// TIA Portal V15.1 export
// export: Created 2024-05-17T05:38:54.9561831Z, ExportSetting WithDefaults, DisplayName Totally Integrated Automation Portal, DisplayVersion V15.1 Update 5, DisplayName TIA Portal Openness, DisplayVersion V15.1 Update 5, DisplayName SINAMICS Startdrive Advanced, DisplayVersion V15.1, DisplayName G130, G150, S120, S150, SINAMICS MV, S210, DisplayVersion V15.1, DisplayName G110M, G120, G120C, G120D, G120P, DisplayVersion V15.1, DisplayName STEP 7 Professional, DisplayVersion V15.1 Update 5, DisplayName STEP 7 Safety, DisplayVersion V15.1, DisplayName WinCC Professional, DisplayVersion V15.1 Update 5, DisplayName SIMATIC Visualization Architect, DisplayVersion V15.1
FUNCTION "209220ZM01" : Void   // FC350, FBD
TITLE = 209220ZM01 ModeZone
{ S7_Optimized_Access := 'FALSE' }
AUTHOR : VCG
NAME : Mot001
VERSION : 0.1
// stored: AutoNumber false, IsIECCheckEnabled false, SetENOAutomatically False, UDAEnableTagReadback false
   VAR_OUTPUT
      O_AlarmA : Bool;   // Alarm A
      O_AlarmB : Bool;   // Alarm B
      O_AlarmC : Bool;   // Alarm C
      O_AlarmD : Bool;   // Alarm D
      O_AlarmABCondition : Bool;   // Alarms resetable
      H_IAnim : Word;   // Animation bits to Icon in WinCC
   END_VAR
   VAR_TEMP
      TempReal : Real;
      TempInt : Int;
   END_VAR
   VAR_TEMP   // added for the SCL form of the ladder/FBD networks
      _w1 : Bool;
      _w2 : Bool;
   END_VAR
BEGIN

REGION Network 1: **** 1 - Inputs **** HMI Commands
   // HMI Commands from the WinCC
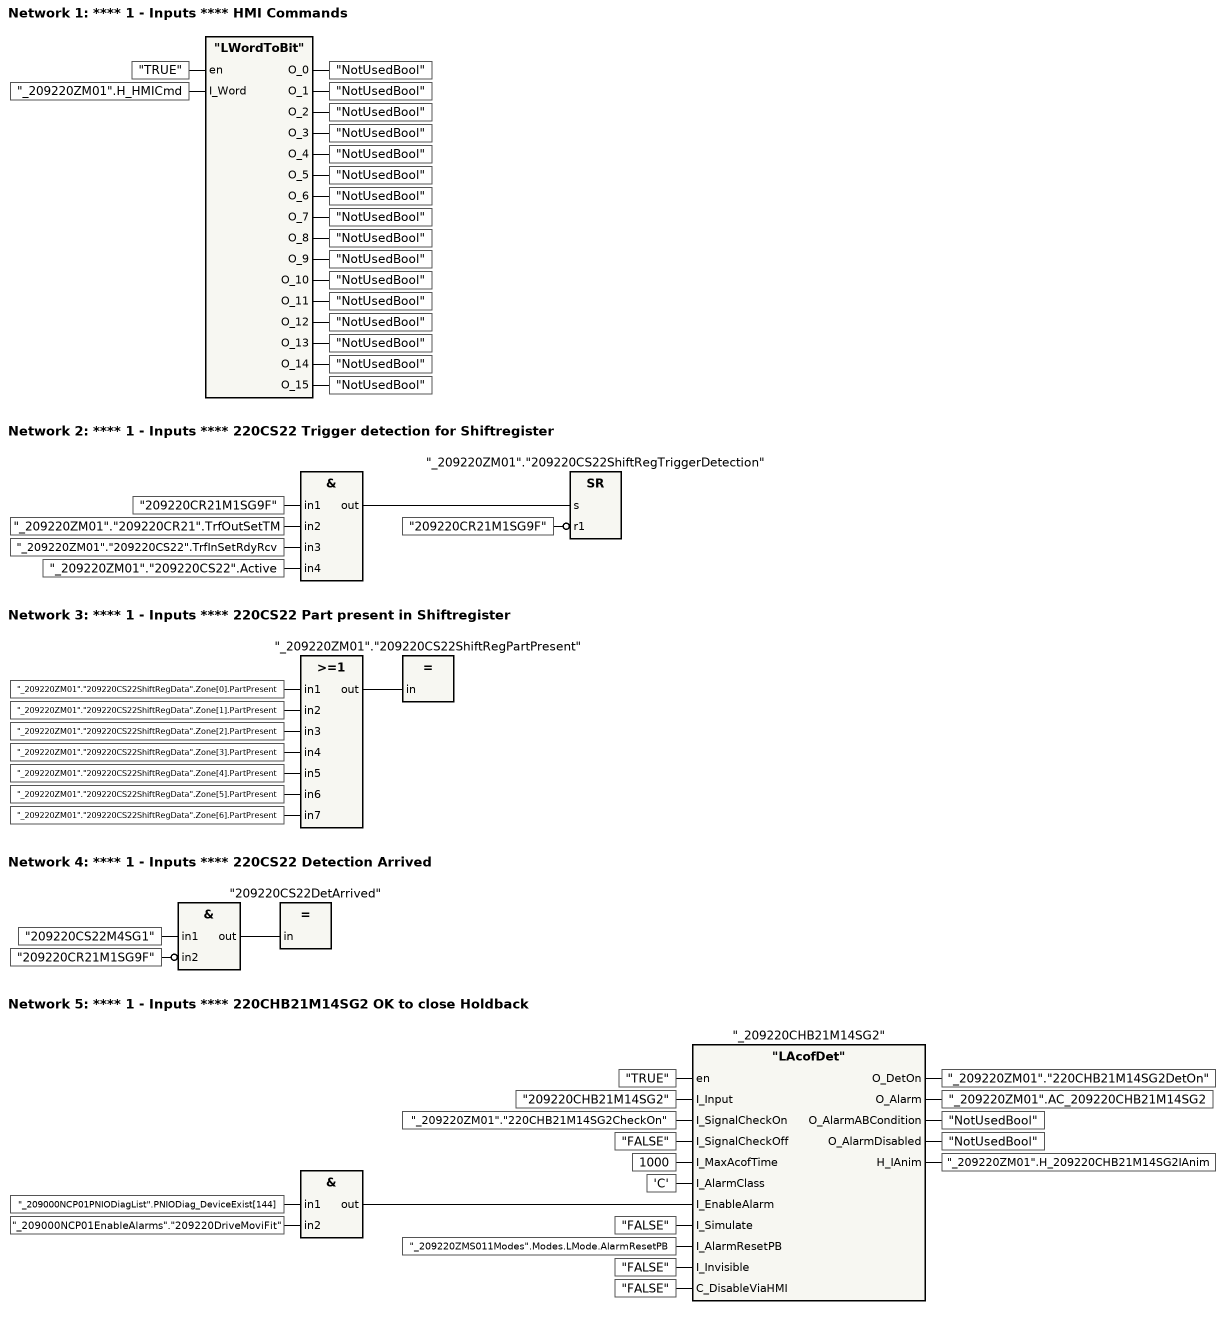
   IF "TRUE" THEN
       "LWordToBit"(I_Word := "_209220ZM01".H_HMICmd,
                    O_0 => "NotUsedBool",
                    O_1 => "NotUsedBool",
                    O_2 => "NotUsedBool",
                    O_3 => "NotUsedBool",
                    O_4 => "NotUsedBool",
                    O_5 => "NotUsedBool",
                    O_6 => "NotUsedBool",
                    O_7 => "NotUsedBool",
                    O_8 => "NotUsedBool",
                    O_9 => "NotUsedBool",
                    O_10 => "NotUsedBool",
                    O_11 => "NotUsedBool",
                    O_12 => "NotUsedBool",
                    O_13 => "NotUsedBool",
                    O_14 => "NotUsedBool",
                    O_15 => "NotUsedBool");
   END_IF;
END_REGION

REGION Network 2: **** 1 - Inputs **** 220CS22 Trigger detection for Shiftregister
   IF "209220CR21M1SG9F" AND "_209220ZM01"."209220CR21".TrfOutSetTM AND "_209220ZM01"."209220CS22".TrfInSetRdyRcv AND "_209220ZM01"."209220CS22".Active THEN
       "_209220ZM01"."209220CS22ShiftRegTriggerDetection" := TRUE;   // SR flip-flop
   END_IF;
   IF NOT "209220CR21M1SG9F" THEN "_209220ZM01"."209220CS22ShiftRegTriggerDetection" := FALSE; END_IF;
END_REGION

REGION Network 3: **** 1 - Inputs **** 220CS22 Part present in Shiftregister
   "_209220ZM01"."209220CS22ShiftRegPartPresent" := "_209220ZM01"."209220CS22ShiftRegData".Zone[0].PartPresent OR "_209220ZM01"."209220CS22ShiftRegData".Zone[1].PartPresent OR "_209220ZM01"."209220CS22ShiftRegData".Zone[2].PartPresent OR "_209220ZM01"."209220CS22ShiftRegData".Zone[3].PartPresent OR "_209220ZM01"."209220CS22ShiftRegData".Zone[4].PartPresent OR "_209220ZM01"."209220CS22ShiftRegData".Zone[5].PartPresent OR "_209220ZM01"."209220CS22ShiftRegData".Zone[6].PartPresent;
END_REGION

REGION Network 4: **** 1 - Inputs **** 220CS22 Detection Arrived
   "209220CS22DetArrived" := "209220CS22M4SG1" AND NOT "209220CR21M1SG9F";
END_REGION

REGION Network 5: **** 1 - Inputs **** 220CHB21M14SG2 OK to close Holdback
   IF "TRUE" THEN
       "_209220CHB21M14SG2"(I_Input := "209220CHB21M14SG2",   // "LAcofDet"
                            I_SignalCheckOn := "_209220ZM01"."220CHB21M14SG2CheckOn",
                            I_SignalCheckOff := "FALSE",
                            I_MaxAcofTime := 1000,
                            I_AlarmClass := 'C',
                            I_EnableAlarm := "_209000NCP01PNIODiagList".PNIODiag_DeviceExist[144] AND "_209000NCP01EnableAlarms"."209220DriveMoviFit",
                            I_Simulate := "FALSE",
                            I_AlarmResetPB := "_209220ZMS011Modes".Modes.LMode.AlarmResetPB,
                            I_Invisible := "FALSE",
                            C_DisableViaHMI := "FALSE",
                            O_DetOn => "_209220ZM01"."220CHB21M14SG2DetOn",
                            O_Alarm => "_209220ZM01".AC_209220CHB21M14SG2,
                            O_AlarmABCondition => "NotUsedBool",
                            O_AlarmDisabled => "NotUsedBool",
                            H_IAnim => "_209220ZM01".H_209220CHB21M14SG2IAnim);
   END_IF;
END_REGION

REGION Network 6: **** 1 - Inputs **** 220CS22M4SG40 Open door detection left
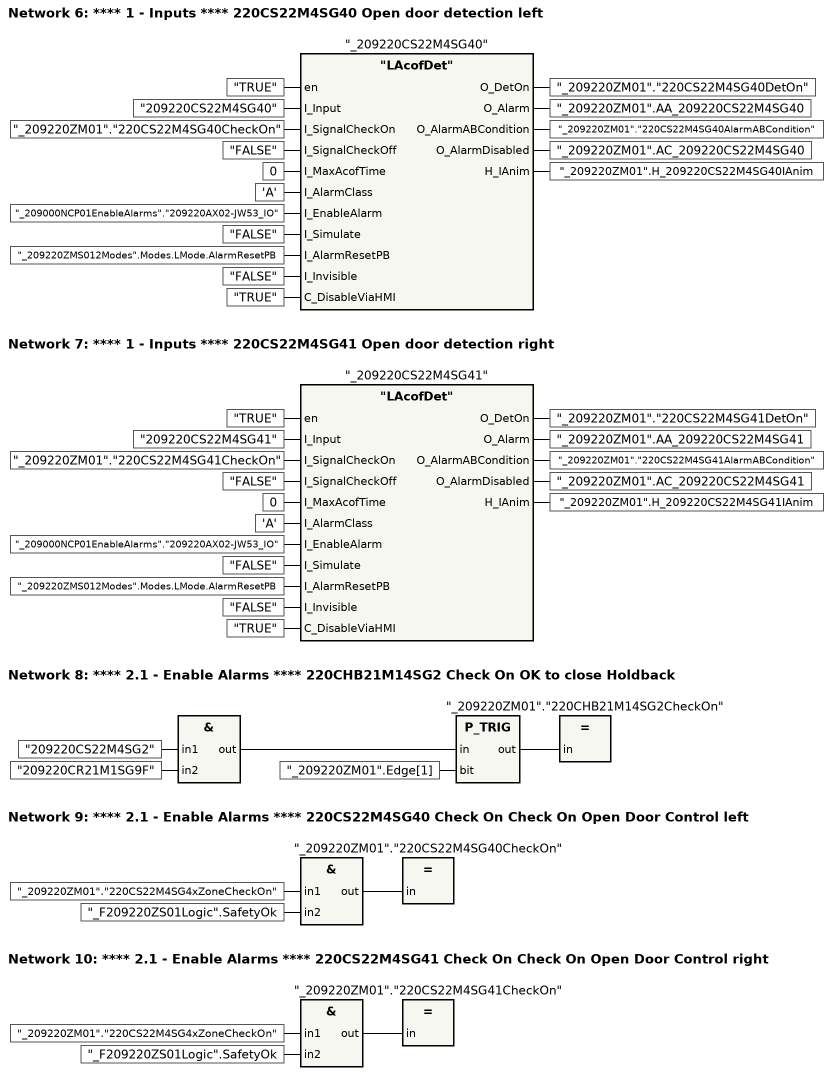
   IF "TRUE" THEN
       "_209220CS22M4SG40"(I_Input := "209220CS22M4SG40",   // "LAcofDet"
                           I_SignalCheckOn := "_209220ZM01"."220CS22M4SG40CheckOn",
                           I_SignalCheckOff := "FALSE",
                           I_MaxAcofTime := 0,
                           I_AlarmClass := 'A',
                           I_EnableAlarm := "_209000NCP01EnableAlarms"."209220AX02-JW53_IO",
                           I_Simulate := "FALSE",
                           I_AlarmResetPB := "_209220ZMS012Modes".Modes.LMode.AlarmResetPB,
                           I_Invisible := "FALSE",
                           C_DisableViaHMI := "TRUE",
                           O_DetOn => "_209220ZM01"."220CS22M4SG40DetOn",
                           O_Alarm => "_209220ZM01".AA_209220CS22M4SG40,
                           O_AlarmABCondition => "_209220ZM01"."220CS22M4SG40AlarmABCondition",
                           O_AlarmDisabled => "_209220ZM01".AC_209220CS22M4SG40,
                           H_IAnim => "_209220ZM01".H_209220CS22M4SG40IAnim);
   END_IF;
END_REGION

REGION Network 7: **** 1 - Inputs **** 220CS22M4SG41 Open door detection right
   IF "TRUE" THEN
       "_209220CS22M4SG41"(I_Input := "209220CS22M4SG41",   // "LAcofDet"
                           I_SignalCheckOn := "_209220ZM01"."220CS22M4SG41CheckOn",
                           I_SignalCheckOff := "FALSE",
                           I_MaxAcofTime := 0,
                           I_AlarmClass := 'A',
                           I_EnableAlarm := "_209000NCP01EnableAlarms"."209220AX02-JW53_IO",
                           I_Simulate := "FALSE",
                           I_AlarmResetPB := "_209220ZMS012Modes".Modes.LMode.AlarmResetPB,
                           I_Invisible := "FALSE",
                           C_DisableViaHMI := "TRUE",
                           O_DetOn => "_209220ZM01"."220CS22M4SG41DetOn",
                           O_Alarm => "_209220ZM01".AA_209220CS22M4SG41,
                           O_AlarmABCondition => "_209220ZM01"."220CS22M4SG41AlarmABCondition",
                           O_AlarmDisabled => "_209220ZM01".AC_209220CS22M4SG41,
                           H_IAnim => "_209220ZM01".H_209220CS22M4SG41IAnim);
   END_IF;
END_REGION

REGION Network 8: **** 2.1 - Enable Alarms **** 220CHB21M14SG2 Check On OK to close Holdback
   #_w1 := "209220CS22M4SG2" AND "209220CR21M1SG9F";
   #_w2 := #_w1 AND NOT "_209220ZM01".Edge[1];   // rising edge
   "_209220ZM01".Edge[1] := #_w1;
   "_209220ZM01"."220CHB21M14SG2CheckOn" := #_w2;
END_REGION

REGION Network 9: **** 2.1 - Enable Alarms **** 220CS22M4SG40 Check On Check On Open Door Control left
   "_209220ZM01"."220CS22M4SG40CheckOn" := "_209220ZM01"."220CS22M4SG4xZoneCheckOn" AND "_F209220ZS01Logic".SafetyOk;
END_REGION

REGION Network 10: **** 2.1 - Enable Alarms **** 220CS22M4SG41 Check On Check On Open Door Control right
   "_209220ZM01"."220CS22M4SG41CheckOn" := "_209220ZM01"."220CS22M4SG4xZoneCheckOn" AND "_F209220ZS01Logic".SafetyOk;
END_REGION

REGION Network 11: **** 3.1 - Communication - Other Systems **** Supervision
   // Supervision
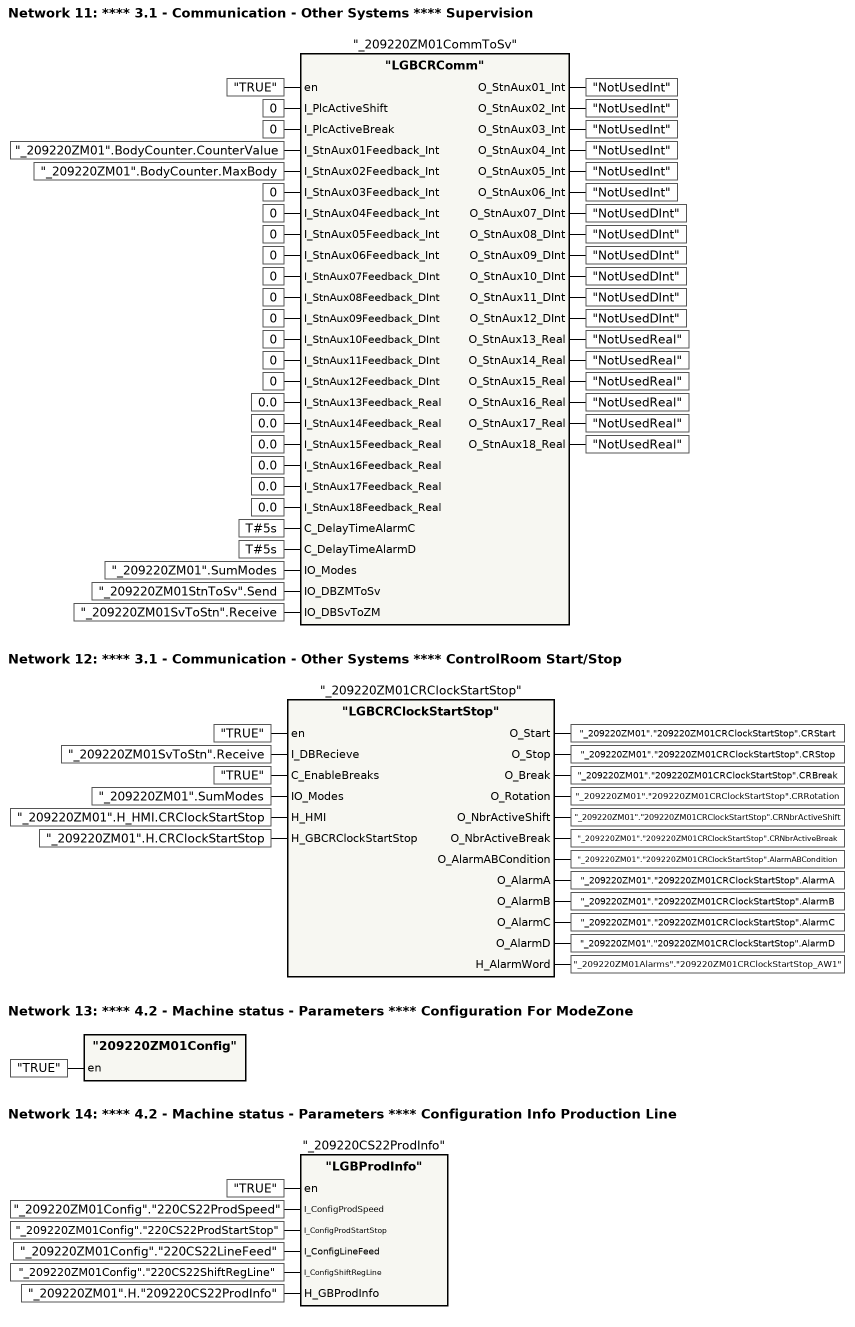
   IF "TRUE" THEN
       "_209220ZM01CommToSv"(I_PlcActiveShift := 0,   // "LGBCRComm"
                             I_PlcActiveBreak := 0,
                             I_StnAux01Feedback_Int := "_209220ZM01".BodyCounter.CounterValue,
                             I_StnAux02Feedback_Int := "_209220ZM01".BodyCounter.MaxBody,
                             I_StnAux03Feedback_Int := 0,
                             I_StnAux04Feedback_Int := 0,
                             I_StnAux05Feedback_Int := 0,
                             I_StnAux06Feedback_Int := 0,
                             I_StnAux07Feedback_DInt := 0,
                             I_StnAux08Feedback_DInt := 0,
                             I_StnAux09Feedback_DInt := 0,
                             I_StnAux10Feedback_DInt := 0,
                             I_StnAux11Feedback_DInt := 0,
                             I_StnAux12Feedback_DInt := 0,
                             I_StnAux13Feedback_Real := 0.0,
                             I_StnAux14Feedback_Real := 0.0,
                             I_StnAux15Feedback_Real := 0.0,
                             I_StnAux16Feedback_Real := 0.0,
                             I_StnAux17Feedback_Real := 0.0,
                             I_StnAux18Feedback_Real := 0.0,
                             C_DelayTimeAlarmC := T#5s,
                             C_DelayTimeAlarmD := T#5s,
                             IO_Modes := "_209220ZM01".SumModes,
                             IO_DBZMToSv := "_209220ZM01StnToSv".Send,
                             IO_DBSvToZM := "_209220ZM01SvToStn".Receive,
                             O_StnAux01_Int => "NotUsedInt",
                             O_StnAux02_Int => "NotUsedInt",
                             O_StnAux03_Int => "NotUsedInt",
                             O_StnAux04_Int => "NotUsedInt",
                             O_StnAux05_Int => "NotUsedInt",
                             O_StnAux06_Int => "NotUsedInt",
                             O_StnAux07_DInt => "NotUsedDInt",
                             O_StnAux08_DInt => "NotUsedDInt",
                             O_StnAux09_DInt => "NotUsedDInt",
                             O_StnAux10_DInt => "NotUsedDInt",
                             O_StnAux11_DInt => "NotUsedDInt",
                             O_StnAux12_DInt => "NotUsedDInt",
                             O_StnAux13_Real => "NotUsedReal",
                             O_StnAux14_Real => "NotUsedReal",
                             O_StnAux15_Real => "NotUsedReal",
                             O_StnAux16_Real => "NotUsedReal",
                             O_StnAux17_Real => "NotUsedReal",
                             O_StnAux18_Real => "NotUsedReal");
   END_IF;
END_REGION

REGION Network 12: **** 3.1 - Communication - Other Systems **** ControlRoom Start/Stop
   IF "TRUE" THEN
       "_209220ZM01CRClockStartStop"(I_DBRecieve := "_209220ZM01SvToStn".Receive,   // "LGBCRClockStartStop"
                               C_EnableBreaks := "TRUE",
                               IO_Modes := "_209220ZM01".SumModes,
                               H_HMI := "_209220ZM01".H_HMI.CRClockStartStop,
                               H_GBCRClockStartStop := "_209220ZM01".H.CRClockStartStop,
                               O_Start => "_209220ZM01"."209220ZM01CRClockStartStop".CRStart,
                               O_Stop => "_209220ZM01"."209220ZM01CRClockStartStop".CRStop,
                               O_Break => "_209220ZM01"."209220ZM01CRClockStartStop".CRBreak,
                               O_Rotation => "_209220ZM01"."209220ZM01CRClockStartStop".CRRotation,
                               O_NbrActiveShift => "_209220ZM01"."209220ZM01CRClockStartStop".CRNbrActiveShift,
                               O_NbrActiveBreak => "_209220ZM01"."209220ZM01CRClockStartStop".CRNbrActiveBreak,
                               O_AlarmABCondition => "_209220ZM01"."209220ZM01CRClockStartStop".AlarmABCondition,
                               O_AlarmA => "_209220ZM01"."209220ZM01CRClockStartStop".AlarmA,
                               O_AlarmB => "_209220ZM01"."209220ZM01CRClockStartStop".AlarmB,
                               O_AlarmC => "_209220ZM01"."209220ZM01CRClockStartStop".AlarmC,
                               O_AlarmD => "_209220ZM01"."209220ZM01CRClockStartStop".AlarmD,
                               H_AlarmWord => "_209220ZM01Alarms"."209220ZM01CRClockStartStop_AW1");
   END_IF;
END_REGION

REGION Network 13: **** 4.2 - Machine status - Parameters **** Configuration For ModeZone
   // Configuration of equipment for ModeZone
   IF "TRUE" THEN "209220ZM01Config"(); END_IF;
END_REGION

REGION Network 14: **** 4.2 - Machine status - Parameters **** Configuration Info Production Line
   IF "TRUE" THEN
       "_209220CS22ProdInfo"(I_ConfigProdSpeed := "_209220ZM01Config"."220CS22ProdSpeed",   // "LGBProdInfo"
                             I_ConfigProdStartStop := "_209220ZM01Config"."220CS22ProdStartStop",
                             I_ConfigLineFeed := "_209220ZM01Config"."220CS22LineFeed",
                             I_ConfigShiftRegLine := "_209220ZM01Config"."220CS22ShiftRegLine",
                             H_GBProdInfo := "_209220ZM01".H."209220CS22ProdInfo");
   END_IF;
END_REGION

REGION Network 15: **** 4.2 - Machine status - Parameters **** Body Counter
   // Body Counter
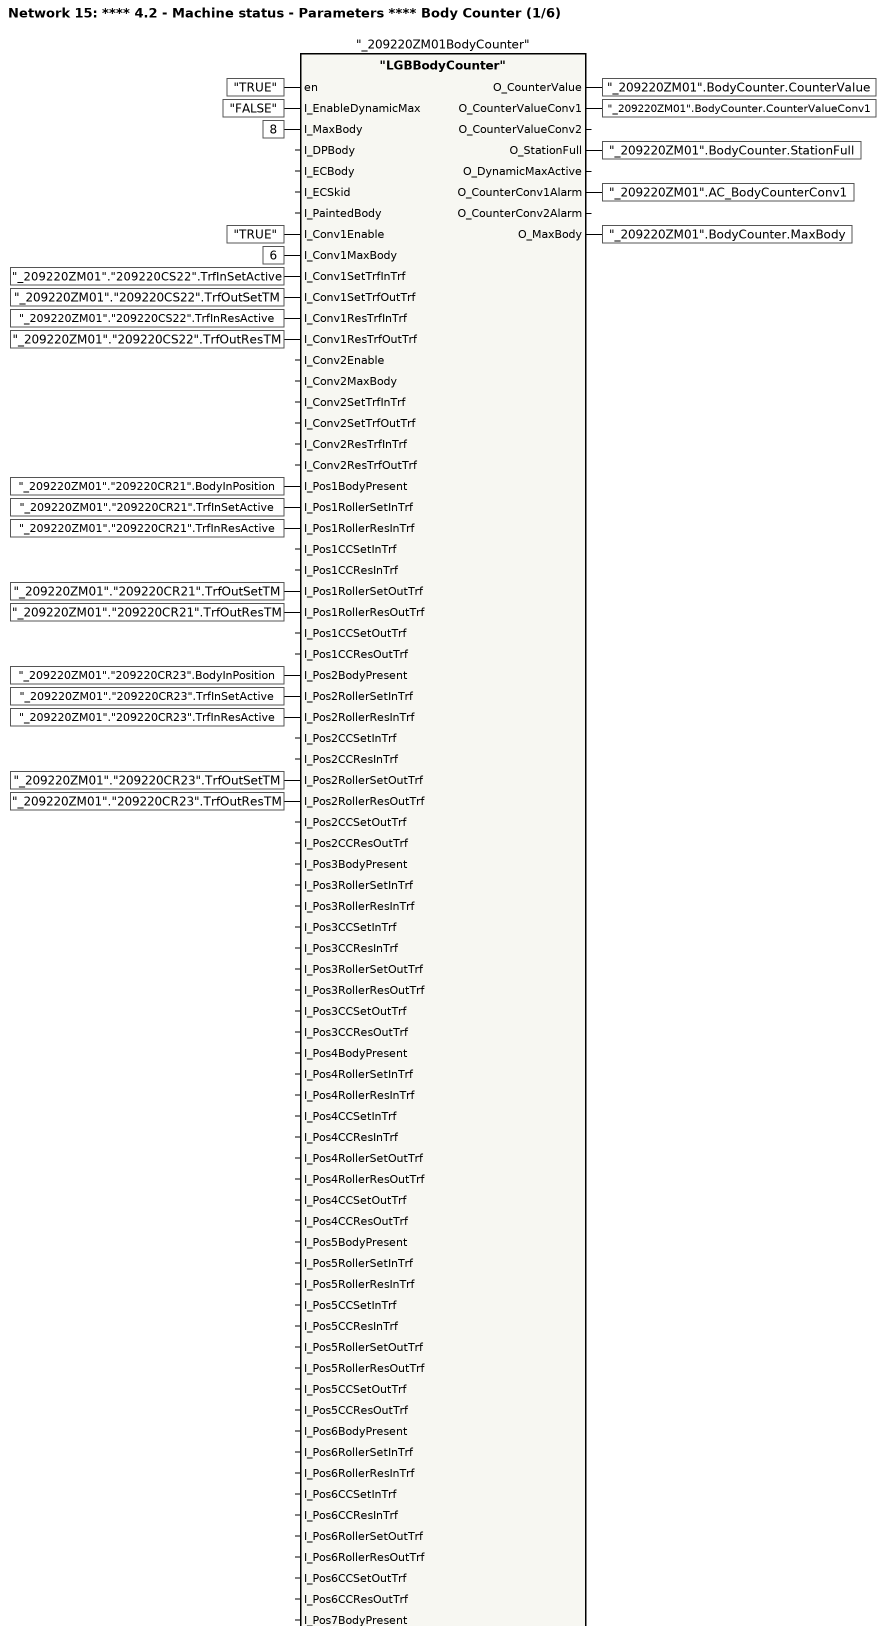
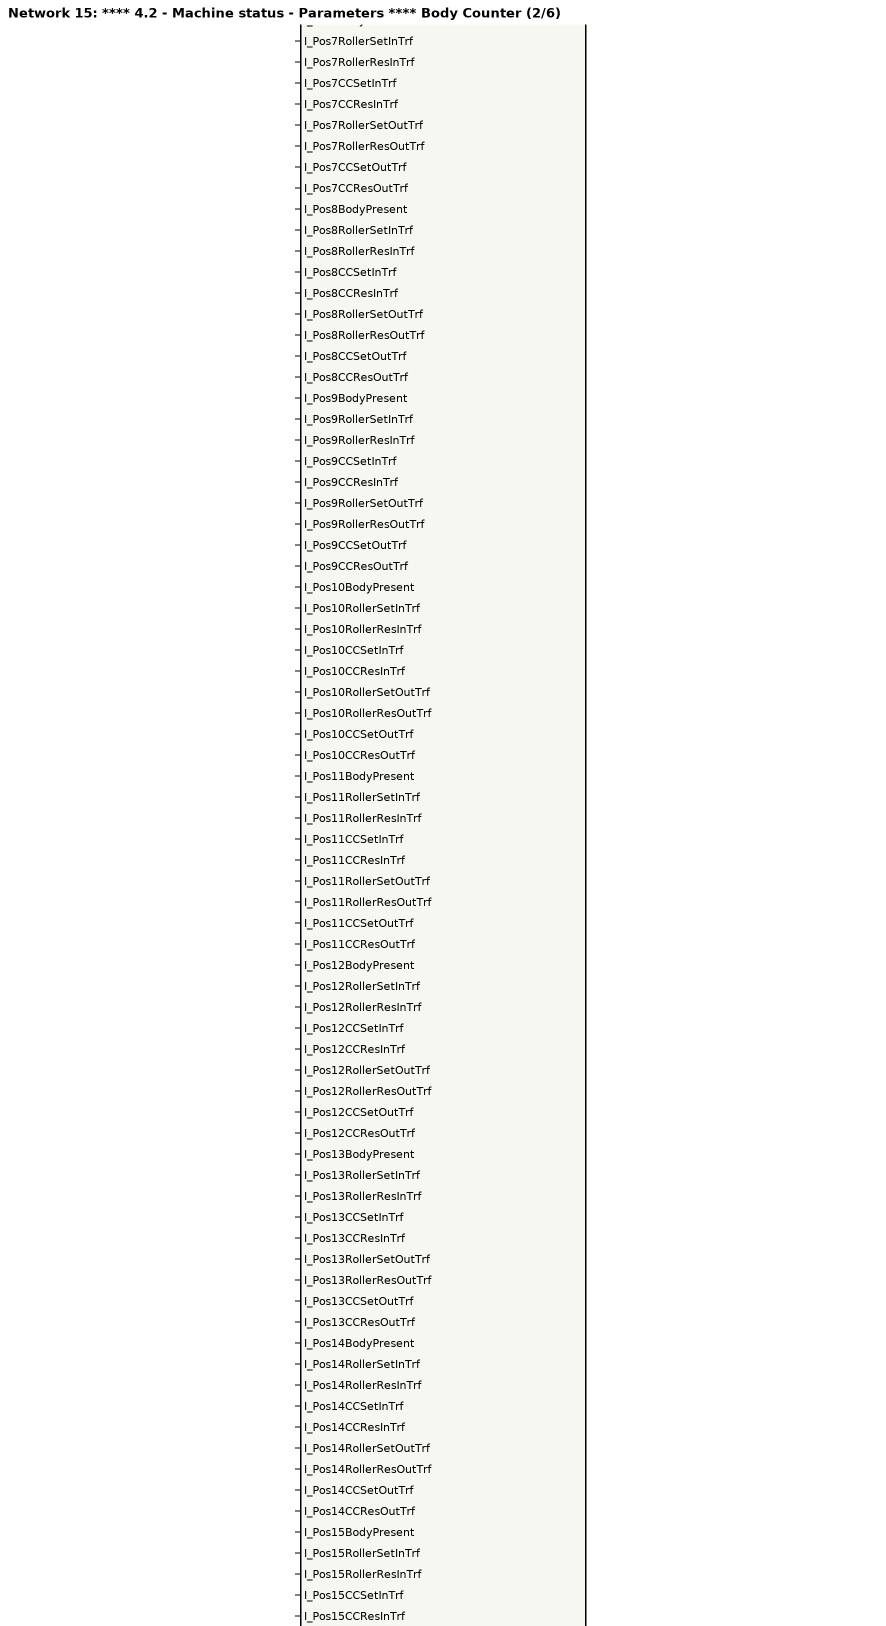
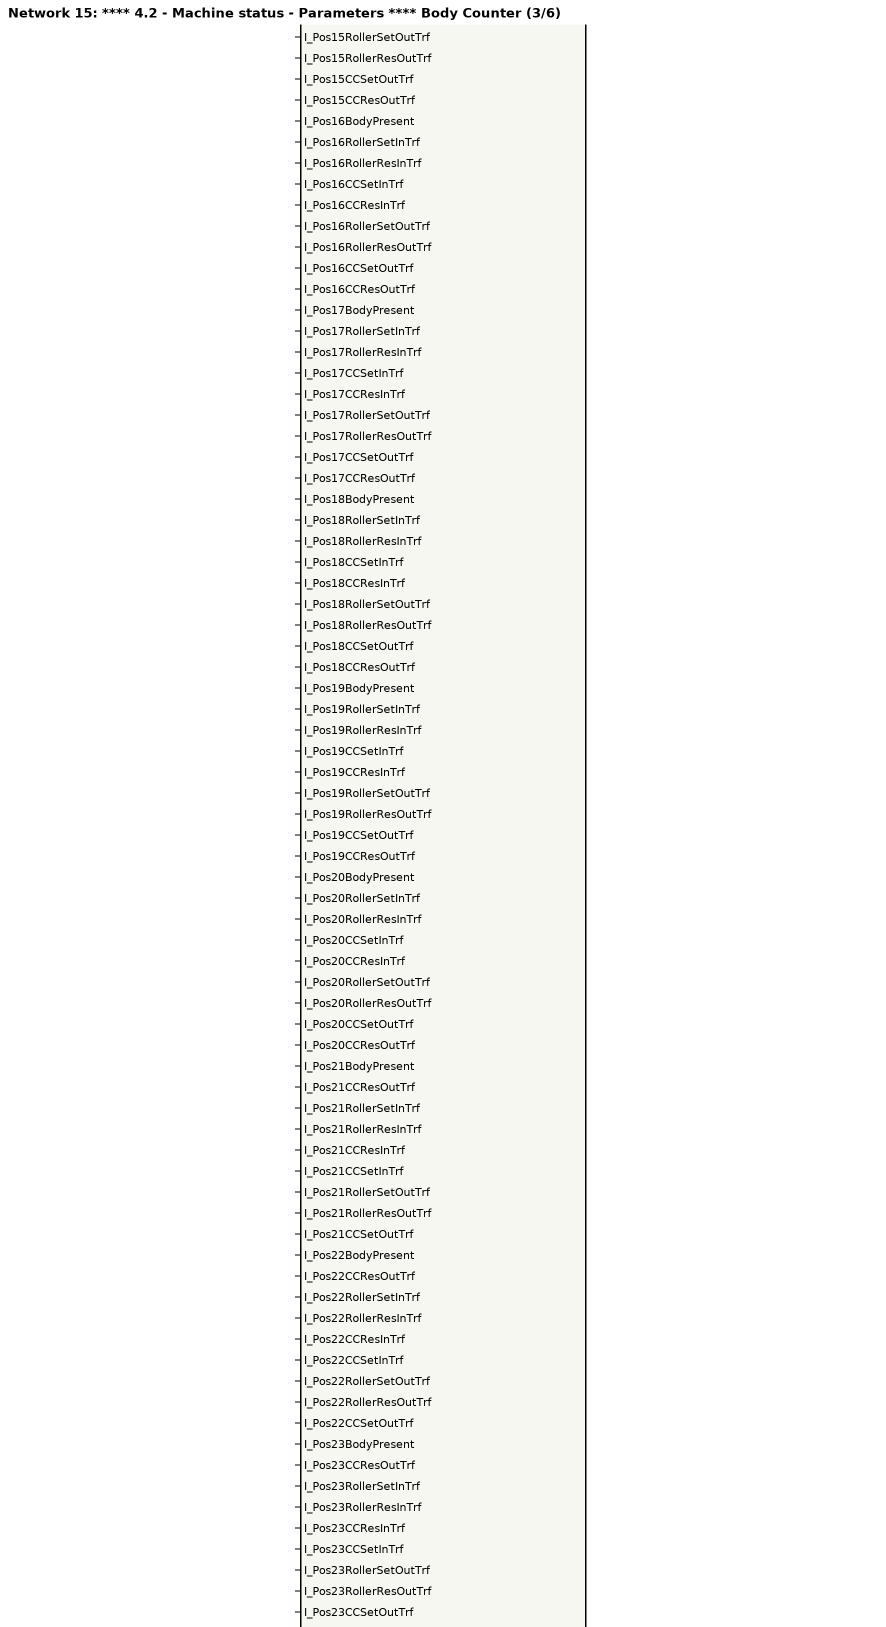
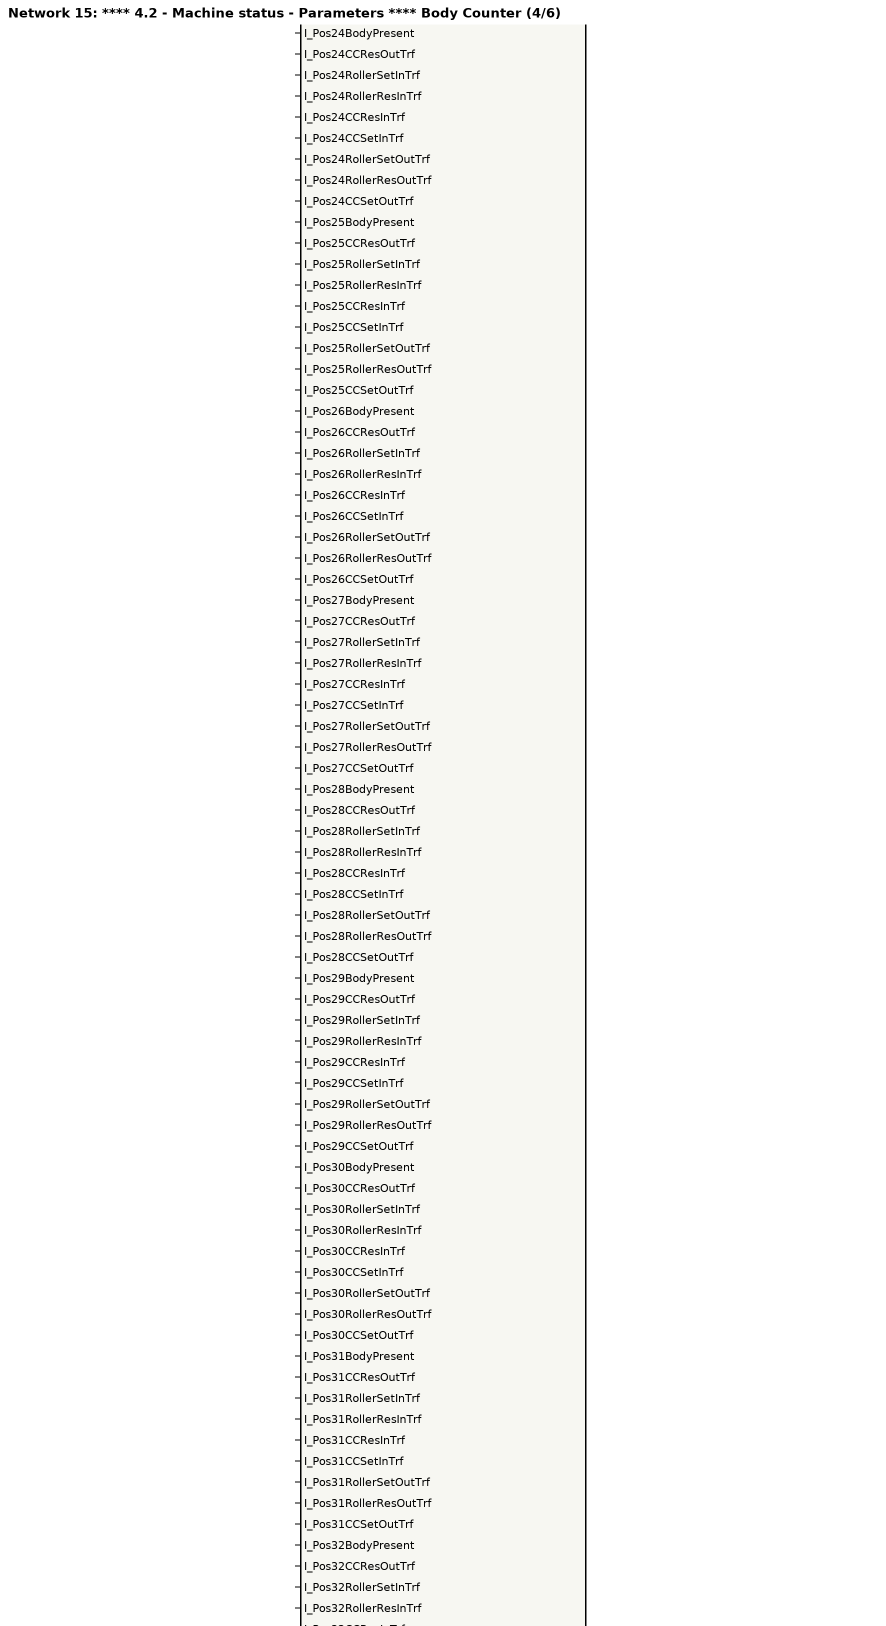
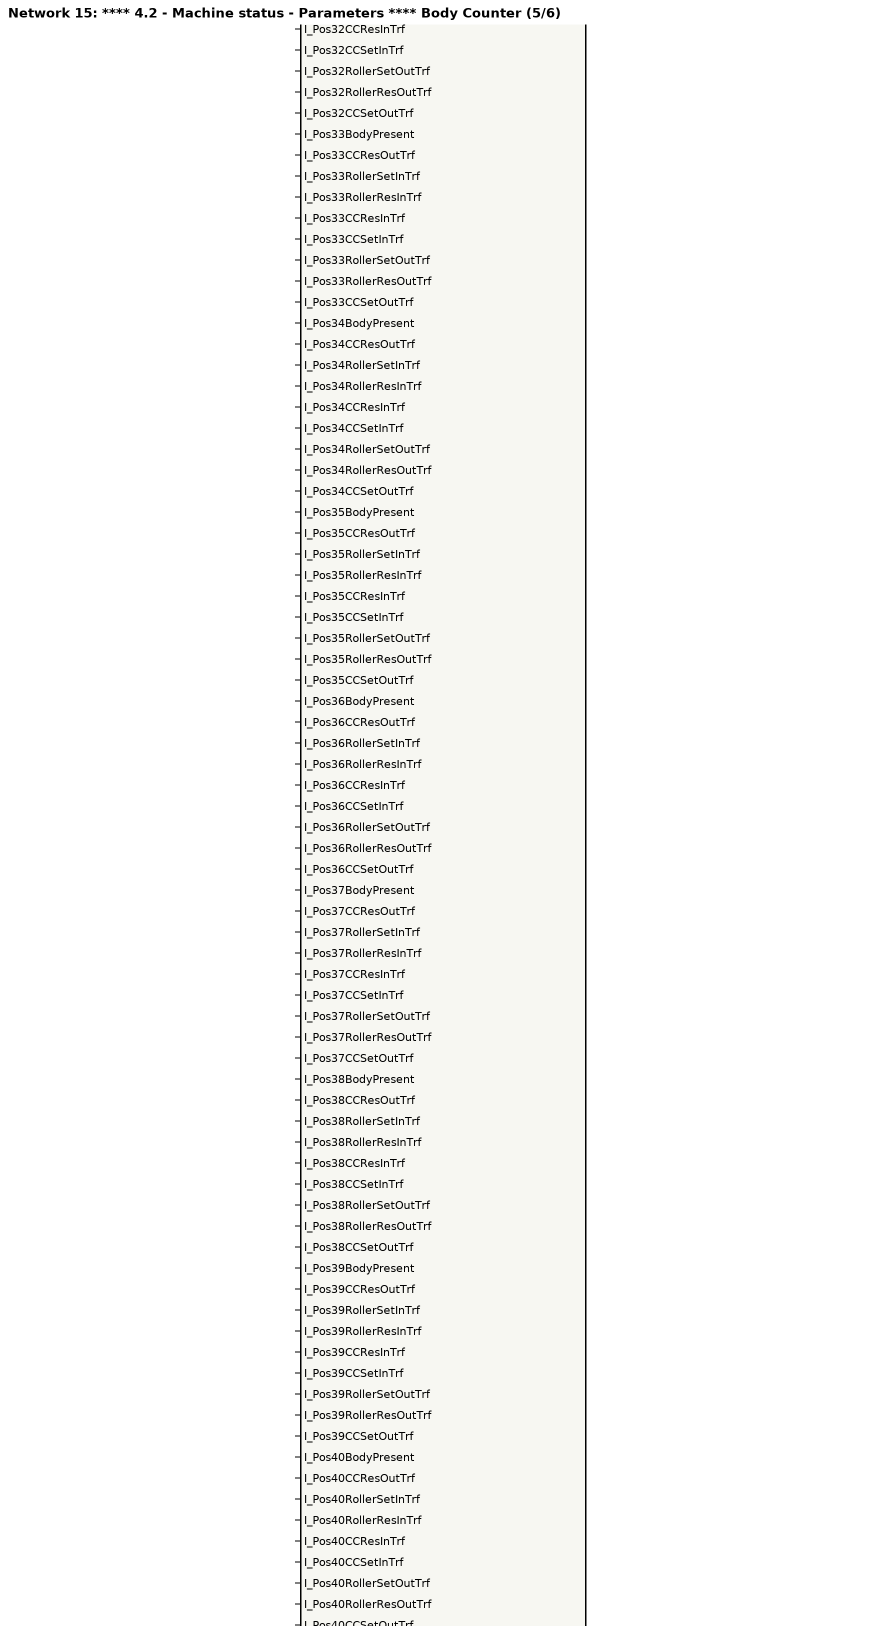
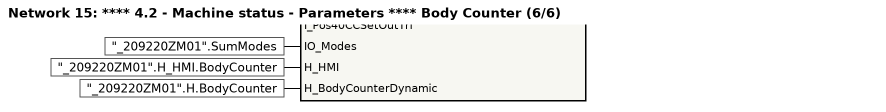
   IF "TRUE" THEN
       "_209220ZM01BodyCounter"(I_EnableDynamicMax := "FALSE",   // "LGBBodyCounter"
                               I_MaxBody := 8,
                               I_Conv1Enable := "TRUE",
                               I_Conv1MaxBody := 6,
                               I_Conv1SetTrfInTrf := "_209220ZM01"."209220CS22".TrfInSetActive,
                               I_Conv1SetTrfOutTrf := "_209220ZM01"."209220CS22".TrfOutSetTM,
                               I_Conv1ResTrfInTrf := "_209220ZM01"."209220CS22".TrfInResActive,
                               I_Conv1ResTrfOutTrf := "_209220ZM01"."209220CS22".TrfOutResTM,
                               I_Pos1BodyPresent := "_209220ZM01"."209220CR21".BodyInPosition,
                               I_Pos1RollerSetInTrf := "_209220ZM01"."209220CR21".TrfInSetActive,
                               I_Pos1RollerResInTrf := "_209220ZM01"."209220CR21".TrfInResActive,
                               I_Pos1RollerSetOutTrf := "_209220ZM01"."209220CR21".TrfOutSetTM,
                               I_Pos1RollerResOutTrf := "_209220ZM01"."209220CR21".TrfOutResTM,
                               I_Pos2BodyPresent := "_209220ZM01"."209220CR23".BodyInPosition,
                               I_Pos2RollerSetInTrf := "_209220ZM01"."209220CR23".TrfInSetActive,
                               I_Pos2RollerResInTrf := "_209220ZM01"."209220CR23".TrfInResActive,
                               I_Pos2RollerSetOutTrf := "_209220ZM01"."209220CR23".TrfOutSetTM,
                               I_Pos2RollerResOutTrf := "_209220ZM01"."209220CR23".TrfOutResTM,
                               IO_Modes := "_209220ZM01".SumModes,
                               H_HMI := "_209220ZM01".H_HMI.BodyCounter,
                               H_BodyCounterDynamic := "_209220ZM01".H.BodyCounter,
                               O_CounterValue => "_209220ZM01".BodyCounter.CounterValue,
                               O_CounterValueConv1 => "_209220ZM01".BodyCounter.CounterValueConv1,
                               O_StationFull => "_209220ZM01".BodyCounter.StationFull,
                               O_CounterConv1Alarm => "_209220ZM01".AC_BodyCounterConv1,
                               O_MaxBody => "_209220ZM01".BodyCounter.MaxBody);
   END_IF;
END_REGION

REGION Network 16: **** 4.4 - Machine Status - Calculation **** 220CS22 Production - Speed
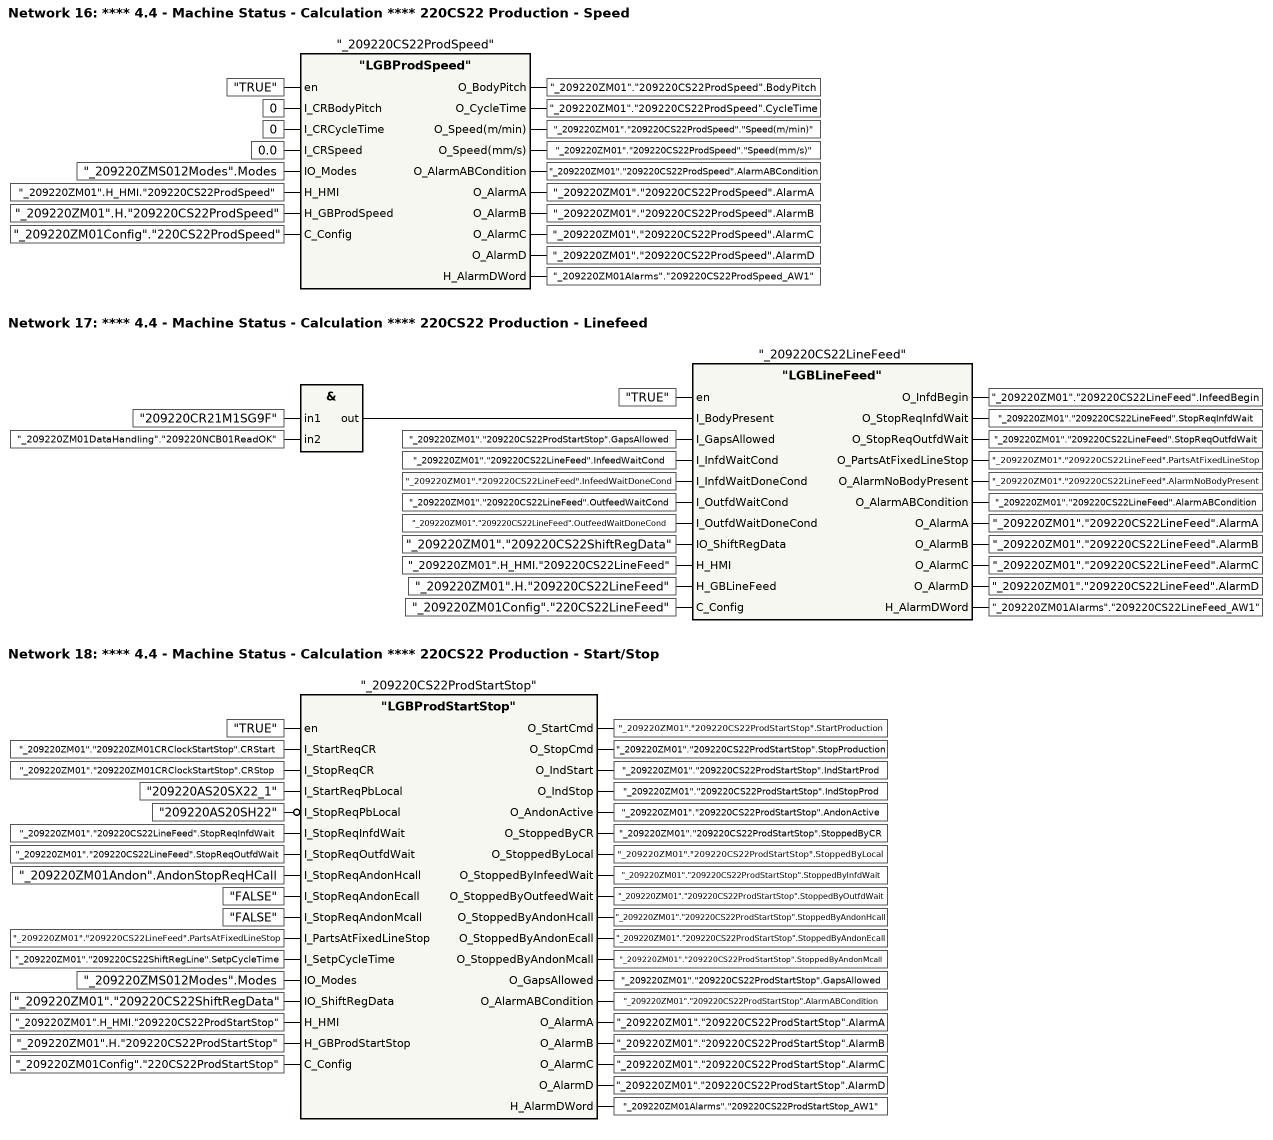
   IF "TRUE" THEN
       "_209220CS22ProdSpeed"(I_CRBodyPitch := 0,   // "LGBProdSpeed"
                              I_CRCycleTime := 0,
                              I_CRSpeed := 0.0,
                              IO_Modes := "_209220ZMS012Modes".Modes,
                              H_HMI := "_209220ZM01".H_HMI."209220CS22ProdSpeed",
                              H_GBProdSpeed := "_209220ZM01".H."209220CS22ProdSpeed",
                              C_Config := "_209220ZM01Config"."220CS22ProdSpeed",
                              O_BodyPitch => "_209220ZM01"."209220CS22ProdSpeed".BodyPitch,
                              O_CycleTime => "_209220ZM01"."209220CS22ProdSpeed".CycleTime,
                              "O_Speed(m/min)" => "_209220ZM01"."209220CS22ProdSpeed"."Speed(m/min)",
                              "O_Speed(mm/s)" => "_209220ZM01"."209220CS22ProdSpeed"."Speed(mm/s)",
                              O_AlarmABCondition => "_209220ZM01"."209220CS22ProdSpeed".AlarmABCondition,
                              O_AlarmA => "_209220ZM01"."209220CS22ProdSpeed".AlarmA,
                              O_AlarmB => "_209220ZM01"."209220CS22ProdSpeed".AlarmB,
                              O_AlarmC => "_209220ZM01"."209220CS22ProdSpeed".AlarmC,
                              O_AlarmD => "_209220ZM01"."209220CS22ProdSpeed".AlarmD,
                              H_AlarmDWord => "_209220ZM01Alarms"."209220CS22ProdSpeed_AW1");
   END_IF;
END_REGION

REGION Network 17: **** 4.4 - Machine Status - Calculation **** 220CS22 Production - Linefeed
   IF "TRUE" THEN
       "_209220CS22LineFeed"(I_BodyPresent := "209220CR21M1SG9F" AND "_209220ZM01DataHandling"."209220NCB01ReadOK",   // "LGBLineFeed"
                             I_GapsAllowed := "_209220ZM01"."209220CS22ProdStartStop".GapsAllowed,
                             I_InfdWaitCond := "_209220ZM01"."209220CS22LineFeed".InfeedWaitCond,
                             I_InfdWaitDoneCond := "_209220ZM01"."209220CS22LineFeed".InfeedWaitDoneCond,
                             I_OutfdWaitCond := "_209220ZM01"."209220CS22LineFeed".OutfeedWaitCond,
                             I_OutfdWaitDoneCond := "_209220ZM01"."209220CS22LineFeed".OutfeedWaitDoneCond,
                             IO_ShiftRegData := "_209220ZM01"."209220CS22ShiftRegData",
                             H_HMI := "_209220ZM01".H_HMI."209220CS22LineFeed",
                             H_GBLineFeed := "_209220ZM01".H."209220CS22LineFeed",
                             C_Config := "_209220ZM01Config"."220CS22LineFeed",
                             O_InfdBegin => "_209220ZM01"."209220CS22LineFeed".InfeedBegin,
                             O_StopReqInfdWait => "_209220ZM01"."209220CS22LineFeed".StopReqInfdWait,
                             O_StopReqOutfdWait => "_209220ZM01"."209220CS22LineFeed".StopReqOutfdWait,
                             O_PartsAtFixedLineStop => "_209220ZM01"."209220CS22LineFeed".PartsAtFixedLineStop,
                             O_AlarmNoBodyPresent => "_209220ZM01"."209220CS22LineFeed".AlarmNoBodyPresent,
                             O_AlarmABCondition => "_209220ZM01"."209220CS22LineFeed".AlarmABCondition,
                             O_AlarmA => "_209220ZM01"."209220CS22LineFeed".AlarmA,
                             O_AlarmB => "_209220ZM01"."209220CS22LineFeed".AlarmB,
                             O_AlarmC => "_209220ZM01"."209220CS22LineFeed".AlarmC,
                             O_AlarmD => "_209220ZM01"."209220CS22LineFeed".AlarmD,
                             H_AlarmDWord => "_209220ZM01Alarms"."209220CS22LineFeed_AW1");
   END_IF;
END_REGION

REGION Network 18: **** 4.4 - Machine Status - Calculation **** 220CS22 Production - Start/Stop
   IF "TRUE" THEN
       "_209220CS22ProdStartStop"(I_StartReqCR := "_209220ZM01"."209220ZM01CRClockStartStop".CRStart,   // "LGBProdStartStop"
                               I_StopReqCR := "_209220ZM01"."209220ZM01CRClockStartStop".CRStop,
                               I_StartReqPbLocal := "209220AS20SX22_1",
                               I_StopReqPbLocal := NOT "209220AS20SH22",
                               I_StopReqInfdWait := "_209220ZM01"."209220CS22LineFeed".StopReqInfdWait,
                               I_StopReqOutfdWait := "_209220ZM01"."209220CS22LineFeed".StopReqOutfdWait,
                               I_StopReqAndonHcall := "_209220ZM01Andon".AndonStopReqHCall,
                               I_StopReqAndonEcall := "FALSE",
                               I_StopReqAndonMcall := "FALSE",
                               I_PartsAtFixedLineStop := "_209220ZM01"."209220CS22LineFeed".PartsAtFixedLineStop,
                               I_SetpCycleTime := "_209220ZM01"."209220CS22ShiftRegLine".SetpCycleTime,
                               IO_Modes := "_209220ZMS012Modes".Modes,
                               IO_ShiftRegData := "_209220ZM01"."209220CS22ShiftRegData",
                               H_HMI := "_209220ZM01".H_HMI."209220CS22ProdStartStop",
                               H_GBProdStartStop := "_209220ZM01".H."209220CS22ProdStartStop",
                               C_Config := "_209220ZM01Config"."220CS22ProdStartStop",
                               O_StartCmd => "_209220ZM01"."209220CS22ProdStartStop".StartProduction,
                               O_StopCmd => "_209220ZM01"."209220CS22ProdStartStop".StopProduction,
                               O_IndStart => "_209220ZM01"."209220CS22ProdStartStop".IndStartProd,
                               O_IndStop => "_209220ZM01"."209220CS22ProdStartStop".IndStopProd,
                               O_AndonActive => "_209220ZM01"."209220CS22ProdStartStop".AndonActive,
                               O_StoppedByCR => "_209220ZM01"."209220CS22ProdStartStop".StoppedByCR,
                               O_StoppedByLocal => "_209220ZM01"."209220CS22ProdStartStop".StoppedByLocal,
                               O_StoppedByInfeedWait => "_209220ZM01"."209220CS22ProdStartStop".StoppedByInfdWait,
                               O_StoppedByOutfeedWait => "_209220ZM01"."209220CS22ProdStartStop".StoppedByOutfdWait,
                               O_StoppedByAndonHcall => "_209220ZM01"."209220CS22ProdStartStop".StoppedByAndonHcall,
                               O_StoppedByAndonEcall => "_209220ZM01"."209220CS22ProdStartStop".StoppedByAndonEcall,
                               O_StoppedByAndonMcall => "_209220ZM01"."209220CS22ProdStartStop".StoppedByAndonMcall,
                               O_GapsAllowed => "_209220ZM01"."209220CS22ProdStartStop".GapsAllowed,
                               O_AlarmABCondition => "_209220ZM01"."209220CS22ProdStartStop".AlarmABCondition,
                               O_AlarmA => "_209220ZM01"."209220CS22ProdStartStop".AlarmA,
                               O_AlarmB => "_209220ZM01"."209220CS22ProdStartStop".AlarmB,
                               O_AlarmC => "_209220ZM01"."209220CS22ProdStartStop".AlarmC,
                               O_AlarmD => "_209220ZM01"."209220CS22ProdStartStop".AlarmD,
                               H_AlarmDWord => "_209220ZM01Alarms"."209220CS22ProdStartStop_AW1");
   END_IF;
END_REGION

REGION Network 19: **** 4.4 - Machine Status - Calculation **** 220CS22 Production - Shiftregister
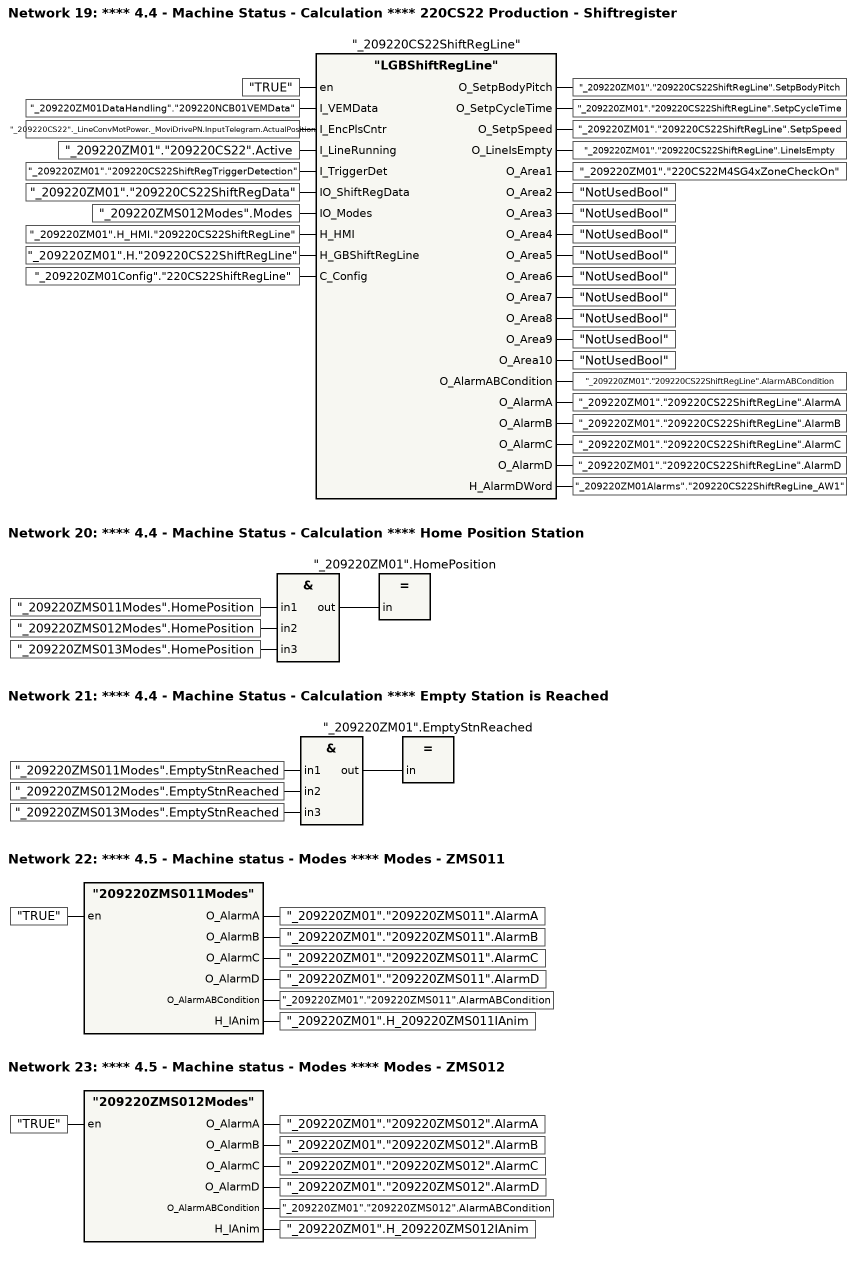
   IF "TRUE" THEN
       "_209220CS22ShiftRegLine"(I_VEMData := "_209220ZM01DataHandling"."209220NCB01VEMData",   // "LGBShiftRegLine"
                               I_EncPlsCntr := "_209220CS22"._LineConvMotPower._MoviDrivePN.InputTelegram.ActualPosition,
                               I_LineRunning := "_209220ZM01"."209220CS22".Active,
                               I_TriggerDet := "_209220ZM01"."209220CS22ShiftRegTriggerDetection",
                               IO_ShiftRegData := "_209220ZM01"."209220CS22ShiftRegData",
                               IO_Modes := "_209220ZMS012Modes".Modes,
                               H_HMI := "_209220ZM01".H_HMI."209220CS22ShiftRegLine",
                               H_GBShiftRegLine := "_209220ZM01".H."209220CS22ShiftRegLine",
                               C_Config := "_209220ZM01Config"."220CS22ShiftRegLine",
                               O_SetpBodyPitch => "_209220ZM01"."209220CS22ShiftRegLine".SetpBodyPitch,
                               O_SetpCycleTime => "_209220ZM01"."209220CS22ShiftRegLine".SetpCycleTime,
                               O_SetpSpeed => "_209220ZM01"."209220CS22ShiftRegLine".SetpSpeed,
                               O_LineIsEmpty => "_209220ZM01"."209220CS22ShiftRegLine".LineIsEmpty,
                               O_Area1 => "_209220ZM01"."220CS22M4SG4xZoneCheckOn",
                               O_Area2 => "NotUsedBool",
                               O_Area3 => "NotUsedBool",
                               O_Area4 => "NotUsedBool",
                               O_Area5 => "NotUsedBool",
                               O_Area6 => "NotUsedBool",
                               O_Area7 => "NotUsedBool",
                               O_Area8 => "NotUsedBool",
                               O_Area9 => "NotUsedBool",
                               O_Area10 => "NotUsedBool",
                               O_AlarmABCondition => "_209220ZM01"."209220CS22ShiftRegLine".AlarmABCondition,
                               O_AlarmA => "_209220ZM01"."209220CS22ShiftRegLine".AlarmA,
                               O_AlarmB => "_209220ZM01"."209220CS22ShiftRegLine".AlarmB,
                               O_AlarmC => "_209220ZM01"."209220CS22ShiftRegLine".AlarmC,
                               O_AlarmD => "_209220ZM01"."209220CS22ShiftRegLine".AlarmD,
                               H_AlarmDWord => "_209220ZM01Alarms"."209220CS22ShiftRegLine_AW1");
   END_IF;
END_REGION

REGION Network 20: **** 4.4 - Machine Status - Calculation **** Home Position Station
   // Home position of the ModeZone
   "_209220ZM01".HomePosition := "_209220ZMS011Modes".HomePosition AND "_209220ZMS012Modes".HomePosition AND "_209220ZMS013Modes".HomePosition;
END_REGION

REGION Network 21: **** 4.4 - Machine Status - Calculation **** Empty Station is Reached
   "_209220ZM01".EmptyStnReached := "_209220ZMS011Modes".EmptyStnReached AND "_209220ZMS012Modes".EmptyStnReached AND "_209220ZMS013Modes".EmptyStnReached;
END_REGION

REGION Network 22: **** 4.5 - Machine status - Modes **** Modes - ZMS011
   // Modes
   IF "TRUE" THEN
       "209220ZMS011Modes"(O_AlarmA => "_209220ZM01"."209220ZMS011".AlarmA,
                           O_AlarmB => "_209220ZM01"."209220ZMS011".AlarmB,
                           O_AlarmC => "_209220ZM01"."209220ZMS011".AlarmC,
                           O_AlarmD => "_209220ZM01"."209220ZMS011".AlarmD,
                           O_AlarmABCondition => "_209220ZM01"."209220ZMS011".AlarmABCondition,
                           H_IAnim => "_209220ZM01".H_209220ZMS011IAnim);
   END_IF;
END_REGION

REGION Network 23: **** 4.5 - Machine status - Modes **** Modes - ZMS012
   // Modes
   IF "TRUE" THEN
       "209220ZMS012Modes"(O_AlarmA => "_209220ZM01"."209220ZMS012".AlarmA,
                           O_AlarmB => "_209220ZM01"."209220ZMS012".AlarmB,
                           O_AlarmC => "_209220ZM01"."209220ZMS012".AlarmC,
                           O_AlarmD => "_209220ZM01"."209220ZMS012".AlarmD,
                           O_AlarmABCondition => "_209220ZM01"."209220ZMS012".AlarmABCondition,
                           H_IAnim => "_209220ZM01".H_209220ZMS012IAnim);
   END_IF;
END_REGION

REGION Network 24: **** 4.5 - Machine status - Modes **** Modes - ZMS013
   // Modes
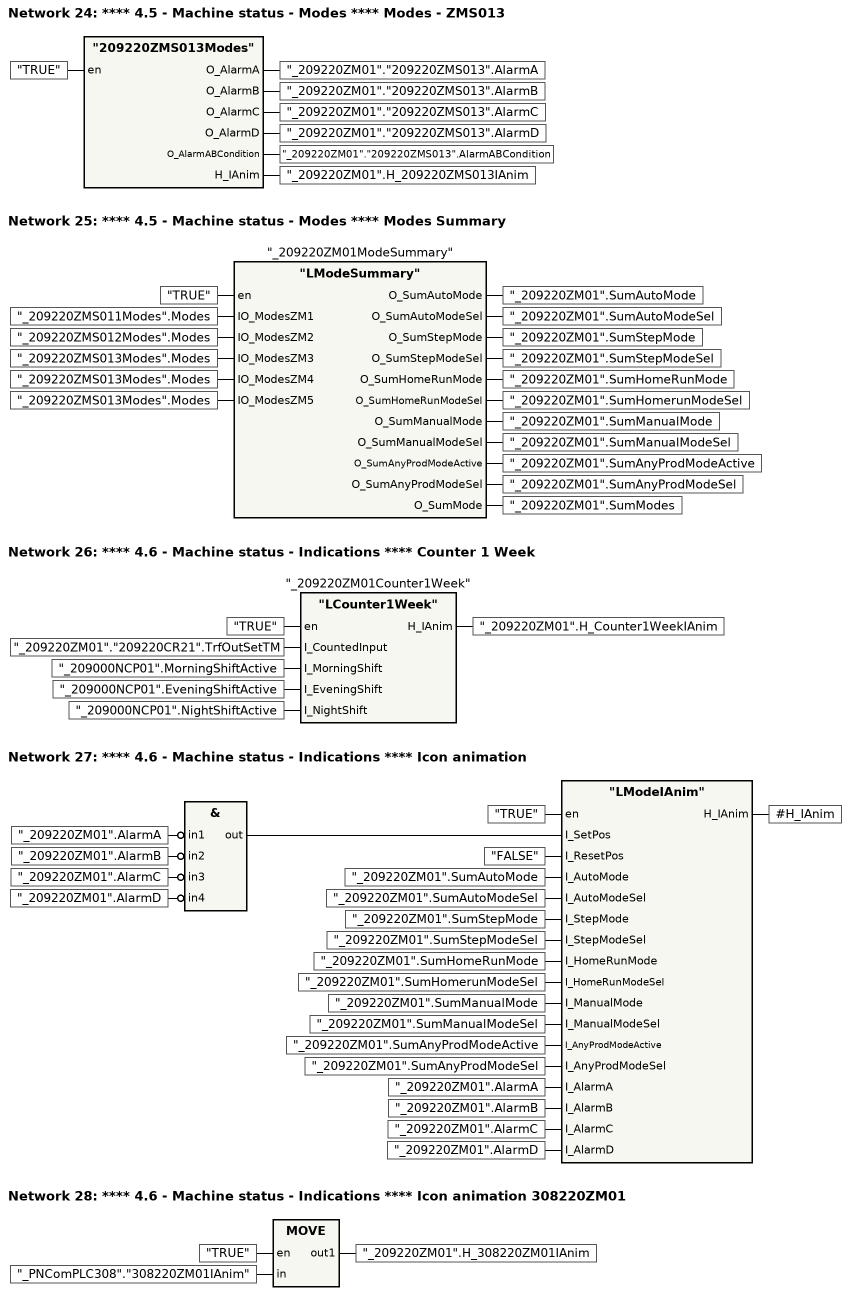
   IF "TRUE" THEN
       "209220ZMS013Modes"(O_AlarmA => "_209220ZM01"."209220ZMS013".AlarmA,
                           O_AlarmB => "_209220ZM01"."209220ZMS013".AlarmB,
                           O_AlarmC => "_209220ZM01"."209220ZMS013".AlarmC,
                           O_AlarmD => "_209220ZM01"."209220ZMS013".AlarmD,
                           O_AlarmABCondition => "_209220ZM01"."209220ZMS013".AlarmABCondition,
                           H_IAnim => "_209220ZM01".H_209220ZMS013IAnim);
   END_IF;
END_REGION

REGION Network 25: **** 4.5 - Machine status - Modes **** Modes Summary
   // Summary of all the modes in safety zone
   IF "TRUE" THEN
       "_209220ZM01ModeSummary"(IO_ModesZM1 := "_209220ZMS011Modes".Modes,   // "LModeSummary"
                               IO_ModesZM2 := "_209220ZMS012Modes".Modes,
                               IO_ModesZM3 := "_209220ZMS013Modes".Modes,
                               IO_ModesZM4 := "_209220ZMS013Modes".Modes,
                               IO_ModesZM5 := "_209220ZMS013Modes".Modes,
                               O_SumAutoMode => "_209220ZM01".SumAutoMode,
                               O_SumAutoModeSel => "_209220ZM01".SumAutoModeSel,
                               O_SumStepMode => "_209220ZM01".SumStepMode,
                               O_SumStepModeSel => "_209220ZM01".SumStepModeSel,
                               O_SumHomeRunMode => "_209220ZM01".SumHomeRunMode,
                               O_SumHomeRunModeSel => "_209220ZM01".SumHomerunModeSel,
                               O_SumManualMode => "_209220ZM01".SumManualMode,
                               O_SumManualModeSel => "_209220ZM01".SumManualModeSel,
                               O_SumAnyProdModeActive => "_209220ZM01".SumAnyProdModeActive,
                               O_SumAnyProdModeSel => "_209220ZM01".SumAnyProdModeSel,
                               O_SumMode => "_209220ZM01".SumModes);
   END_IF;
END_REGION

REGION Network 26: **** 4.6 - Machine status - Indications **** Counter 1 Week
   IF "TRUE" THEN
       "_209220ZM01Counter1Week"(I_CountedInput := "_209220ZM01"."209220CR21".TrfOutSetTM,   // "LCounter1Week"
                               I_MorningShift := "_209000NCP01".MorningShiftActive,
                               I_EveningShift := "_209000NCP01".EveningShiftActive,
                               I_NightShift := "_209000NCP01".NightShiftActive,
                               H_IAnim => "_209220ZM01".H_Counter1WeekIAnim);
   END_IF;
END_REGION

REGION Network 27: **** 4.6 - Machine status - Indications **** Icon animation
   // Icon animation
   IF "TRUE" THEN
       "LModeIAnim"(I_SetPos := NOT "_209220ZM01".AlarmA AND NOT "_209220ZM01".AlarmB AND NOT "_209220ZM01".AlarmC AND NOT "_209220ZM01".AlarmD,
                    I_ResetPos := "FALSE",
                    I_AutoMode := "_209220ZM01".SumAutoMode,
                    I_AutoModeSel := "_209220ZM01".SumAutoModeSel,
                    I_StepMode := "_209220ZM01".SumStepMode,
                    I_StepModeSel := "_209220ZM01".SumStepModeSel,
                    I_HomeRunMode := "_209220ZM01".SumHomeRunMode,
                    I_HomeRunModeSel := "_209220ZM01".SumHomerunModeSel,
                    I_ManualMode := "_209220ZM01".SumManualMode,
                    I_ManualModeSel := "_209220ZM01".SumManualModeSel,
                    I_AnyProdModeActive := "_209220ZM01".SumAnyProdModeActive,
                    I_AnyProdModeSel := "_209220ZM01".SumAnyProdModeSel,
                    I_AlarmA := "_209220ZM01".AlarmA,
                    I_AlarmB := "_209220ZM01".AlarmB,
                    I_AlarmC := "_209220ZM01".AlarmC,
                    I_AlarmD := "_209220ZM01".AlarmD,
                    H_IAnim => #H_IAnim);
   END_IF;
END_REGION

REGION Network 28: **** 4.6 - Machine status - Indications **** Icon animation 308220ZM01
   // Icon animation
   IF "TRUE" THEN "_209220ZM01".H_308220ZM01IAnim := "_PNComPLC308"."308220ZM01IAnim"; END_IF;
END_REGION

REGION Network 29: **** 4.6 - Machine status - Indications **** Icon animation 212A
   // Icon animation
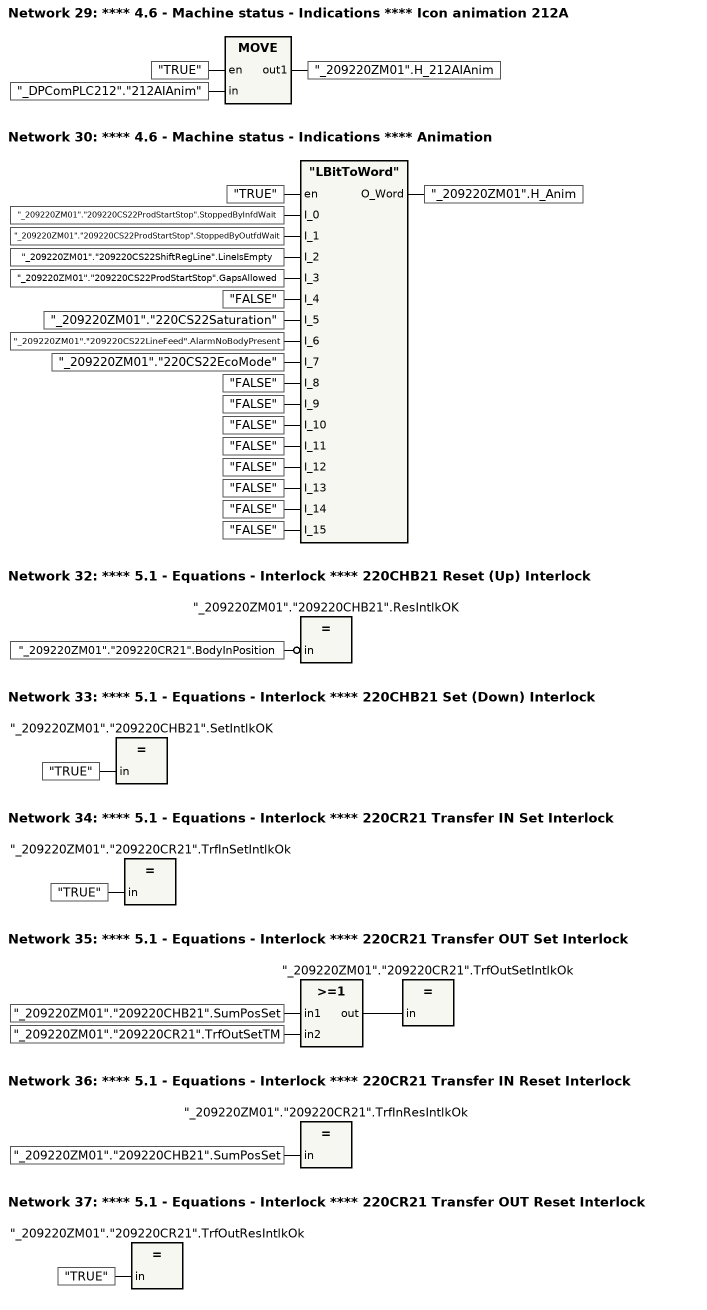
   IF "TRUE" THEN "_209220ZM01".H_212AIAnim := "_DPComPLC212"."212AIAnim"; END_IF;
END_REGION

REGION Network 30: **** 4.6 - Machine status - Indications **** Animation
   // Animation
   IF "TRUE" THEN
       "LBitToWord"(I_0 := "_209220ZM01"."209220CS22ProdStartStop".StoppedByInfdWait,
                    I_1 := "_209220ZM01"."209220CS22ProdStartStop".StoppedByOutfdWait,
                    I_2 := "_209220ZM01"."209220CS22ShiftRegLine".LineIsEmpty,
                    I_3 := "_209220ZM01"."209220CS22ProdStartStop".GapsAllowed,
                    I_4 := "FALSE",
                    I_5 := "_209220ZM01"."220CS22Saturation",
                    I_6 := "_209220ZM01"."209220CS22LineFeed".AlarmNoBodyPresent,
                    I_7 := "_209220ZM01"."220CS22EcoMode",
                    I_8 := "FALSE",
                    I_9 := "FALSE",
                    I_10 := "FALSE",
                    I_11 := "FALSE",
                    I_12 := "FALSE",
                    I_13 := "FALSE",
                    I_14 := "FALSE",
                    I_15 := "FALSE",
                    O_Word => "_209220ZM01".H_Anim);
   END_IF;
END_REGION

NETWORK
TITLE = **** 4.6 - Machine Status - Indications **** Animation DB number
// DB number
      OPN   "_209220ZM01";
      L     DBNO;
      T     "_209220ZM01".H_DBnr;

REGION Network 32: **** 5.1 - Equations - Interlock **** 220CHB21 Reset (Up) Interlock
   "_209220ZM01"."209220CHB21".ResIntlkOK := NOT "_209220ZM01"."209220CR21".BodyInPosition;
END_REGION

REGION Network 33: **** 5.1 - Equations - Interlock **** 220CHB21 Set (Down) Interlock
   "_209220ZM01"."209220CHB21".SetIntlkOK := "TRUE";
END_REGION

REGION Network 34: **** 5.1 - Equations - Interlock **** 220CR21 Transfer IN Set Interlock
   "_209220ZM01"."209220CR21".TrfInSetIntlkOk := "TRUE";
END_REGION

REGION Network 35: **** 5.1 - Equations - Interlock **** 220CR21 Transfer OUT Set Interlock
   "_209220ZM01"."209220CR21".TrfOutSetIntlkOk := "_209220ZM01"."209220CHB21".SumPosSet OR "_209220ZM01"."209220CR21".TrfOutSetTM;
END_REGION

REGION Network 36: **** 5.1 - Equations - Interlock **** 220CR21 Transfer IN Reset Interlock
   "_209220ZM01"."209220CR21".TrfInResIntlkOk := "_209220ZM01"."209220CHB21".SumPosSet;
END_REGION

REGION Network 37: **** 5.1 - Equations - Interlock **** 220CR21 Transfer OUT Reset Interlock
   "_209220ZM01"."209220CR21".TrfOutResIntlkOk := "TRUE";
END_REGION

REGION Network 38: **** 5.1 - Equations - Interlock **** 220CS22 Transfer IN Set Interlock
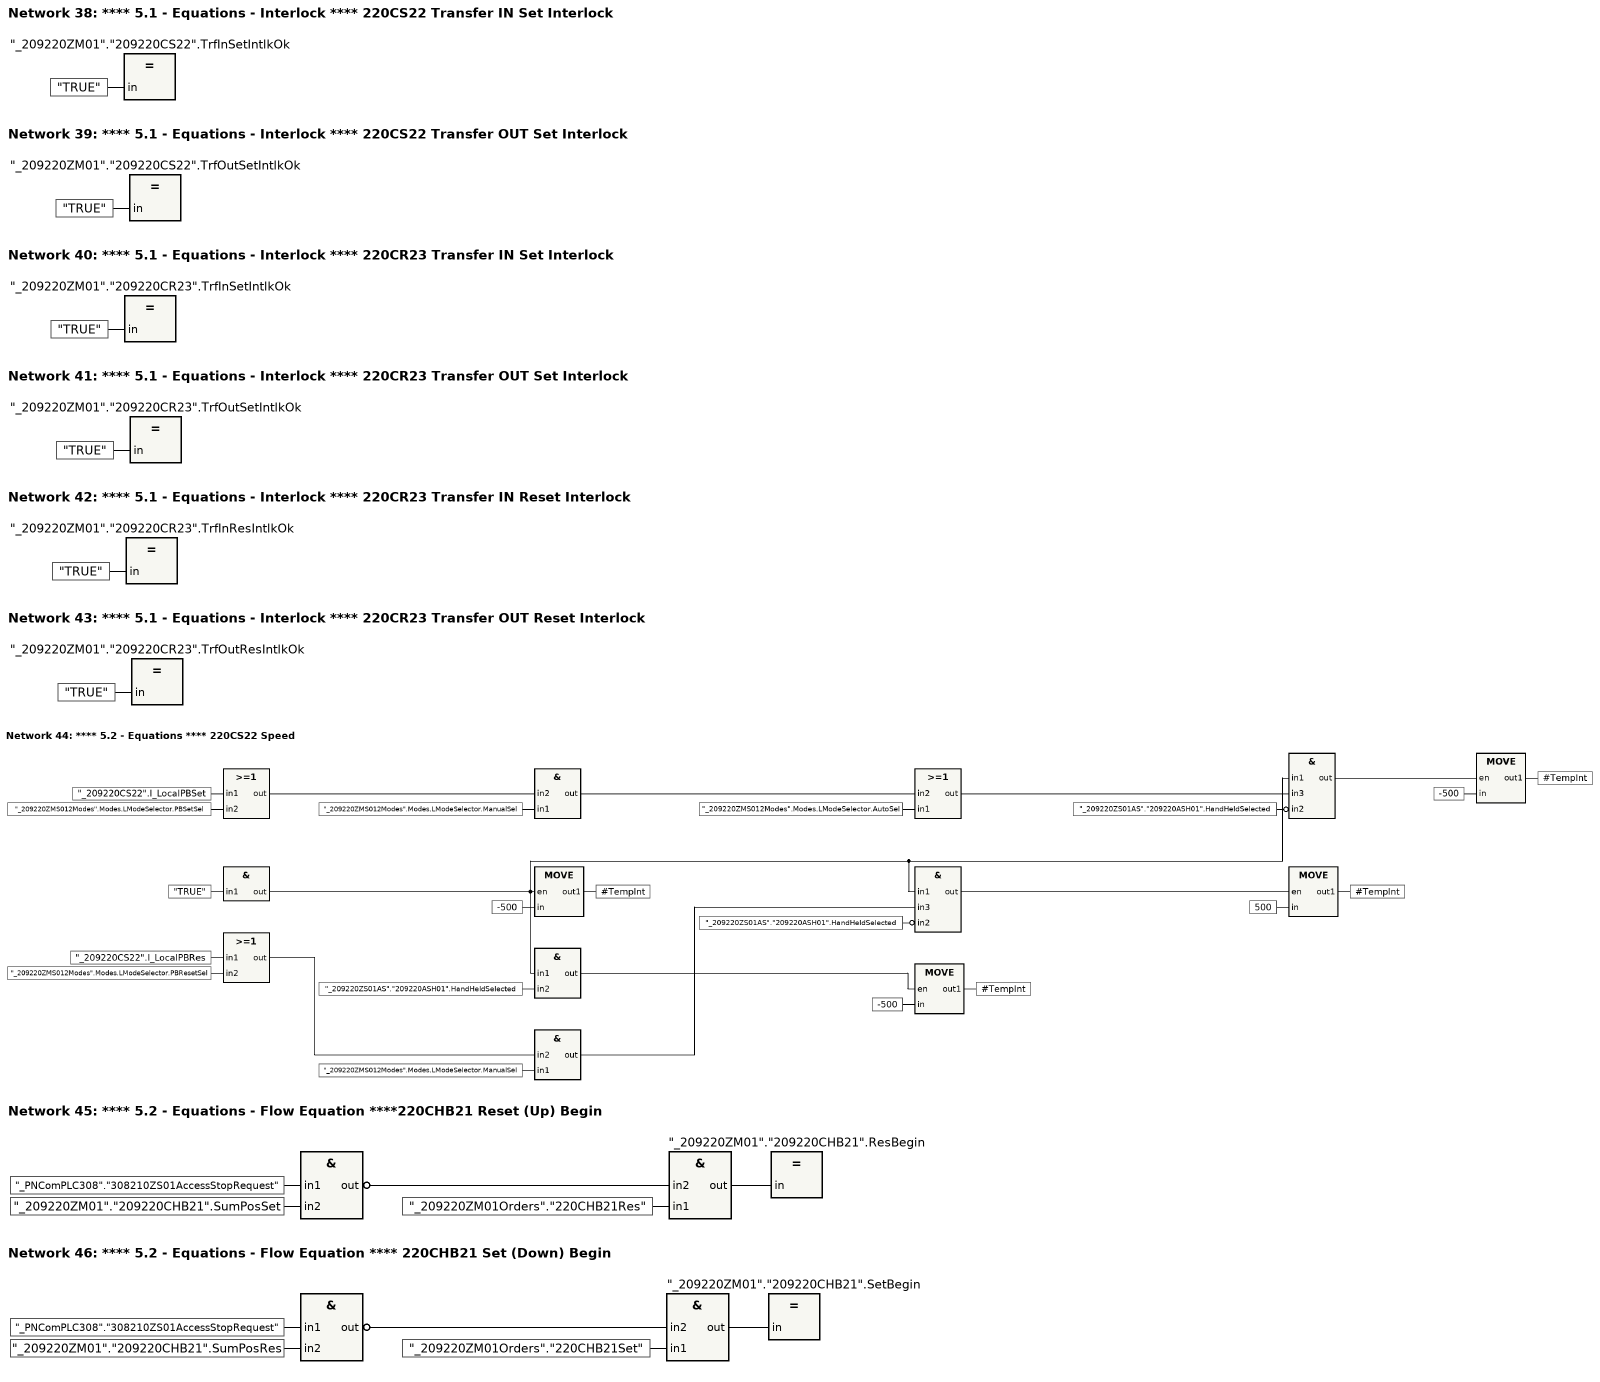
   "_209220ZM01"."209220CS22".TrfInSetIntlkOk := "TRUE";
END_REGION

REGION Network 39: **** 5.1 - Equations - Interlock **** 220CS22 Transfer OUT Set Interlock
   "_209220ZM01"."209220CS22".TrfOutSetIntlkOk := "TRUE";
END_REGION

REGION Network 40: **** 5.1 - Equations - Interlock **** 220CR23 Transfer IN Set Interlock
   "_209220ZM01"."209220CR23".TrfInSetIntlkOk := "TRUE";
END_REGION

REGION Network 41: **** 5.1 - Equations - Interlock **** 220CR23 Transfer OUT Set Interlock
   "_209220ZM01"."209220CR23".TrfOutSetIntlkOk := "TRUE";
END_REGION

REGION Network 42: **** 5.1 - Equations - Interlock **** 220CR23 Transfer IN Reset Interlock
   "_209220ZM01"."209220CR23".TrfInResIntlkOk := "TRUE";
END_REGION

REGION Network 43: **** 5.1 - Equations - Interlock **** 220CR23 Transfer OUT Reset Interlock
   "_209220ZM01"."209220CR23".TrfOutResIntlkOk := "TRUE";
END_REGION

REGION Network 44: **** 5.2 - Equations **** 220CS22 Speed
   IF "TRUE" THEN #TempInt := -500; END_IF;
   IF "TRUE" AND ((("_209220CS22".I_LocalPBSet OR "_209220ZMS012Modes".Modes.LModeSelector.PBSetSel) AND "_209220ZMS012Modes".Modes.LModeSelector.ManualSel) OR "_209220ZMS012Modes".Modes.LModeSelector.AutoSel) AND NOT "_209220ZS01AS"."209220ASH01".HandHeldSelected THEN
       #TempInt := -500;
   END_IF;
   IF "TRUE" AND ("_209220CS22".I_LocalPBRes OR "_209220ZMS012Modes".Modes.LModeSelector.PBResetSel) AND "_209220ZMS012Modes".Modes.LModeSelector.ManualSel AND NOT "_209220ZS01AS"."209220ASH01".HandHeldSelected THEN
       #TempInt := 500;
   END_IF;
   IF "TRUE" AND "_209220ZS01AS"."209220ASH01".HandHeldSelected THEN #TempInt := -500; END_IF;
END_REGION

REGION Network 45: **** 5.2 - Equations - Flow Equation ****220CHB21 Reset (Up) Begin
   "_209220ZM01"."209220CHB21".ResBegin := NOT ("_PNComPLC308"."308210ZS01AccessStopRequest" AND "_209220ZM01"."209220CHB21".SumPosSet) AND "_209220ZM01Orders"."220CHB21Res";
END_REGION

REGION Network 46: **** 5.2 - Equations - Flow Equation **** 220CHB21 Set (Down) Begin
   "_209220ZM01"."209220CHB21".SetBegin := NOT ("_PNComPLC308"."308210ZS01AccessStopRequest" AND "_209220ZM01"."209220CHB21".SumPosRes) AND "_209220ZM01Orders"."220CHB21Set";
END_REGION

REGION Network 47: **** 5.2 - Equations - Flow Equation **** 220CR21 Transfer IN Set Begin
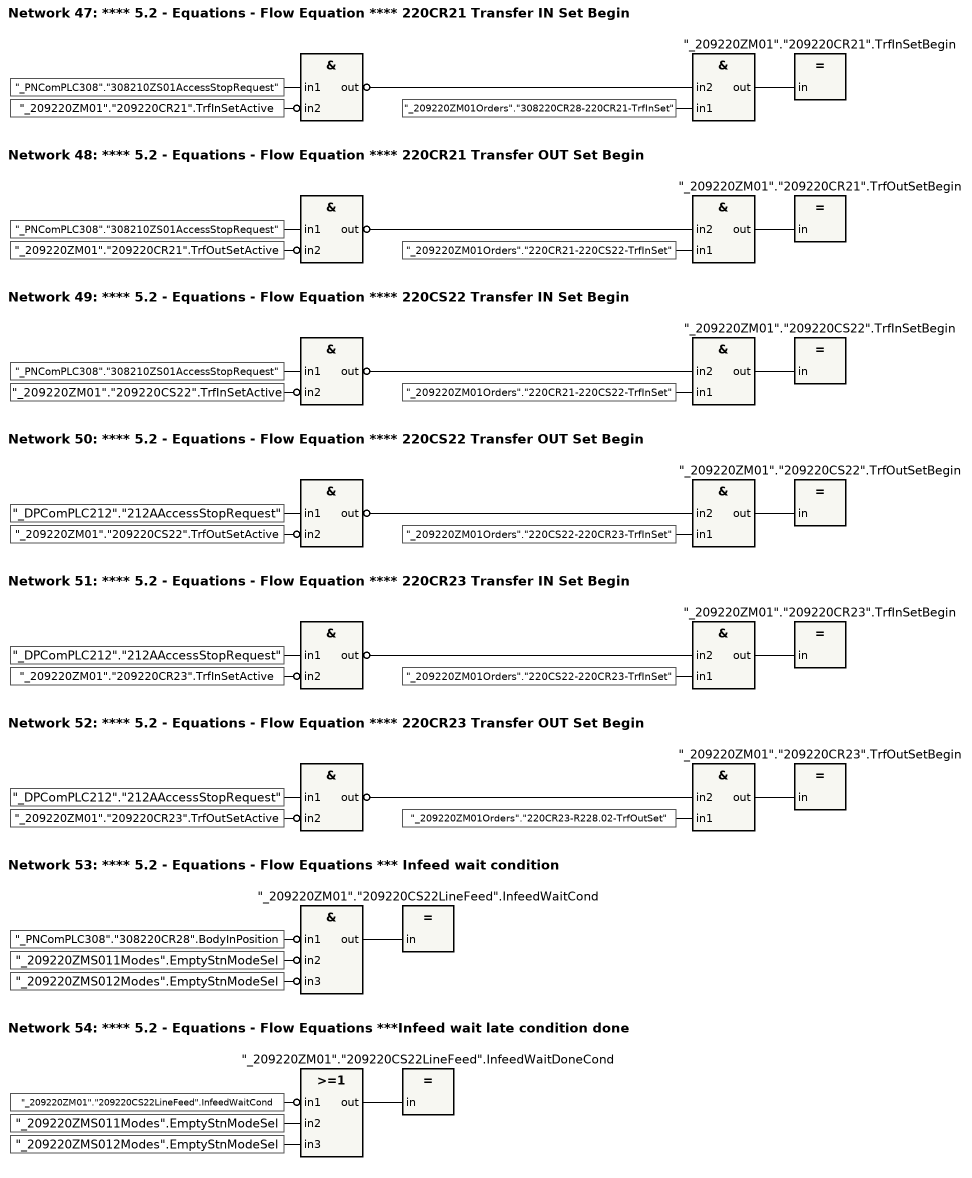
   "_209220ZM01"."209220CR21".TrfInSetBegin := NOT ("_PNComPLC308"."308210ZS01AccessStopRequest" AND NOT "_209220ZM01"."209220CR21".TrfInSetActive) AND "_209220ZM01Orders"."308220CR28-220CR21-TrfInSet";
END_REGION

REGION Network 48: **** 5.2 - Equations - Flow Equation **** 220CR21 Transfer OUT Set Begin
   "_209220ZM01"."209220CR21".TrfOutSetBegin := NOT ("_PNComPLC308"."308210ZS01AccessStopRequest" AND NOT "_209220ZM01"."209220CR21".TrfOutSetActive) AND "_209220ZM01Orders"."220CR21-220CS22-TrfInSet";
END_REGION

REGION Network 49: **** 5.2 - Equations - Flow Equation **** 220CS22 Transfer IN Set Begin
   "_209220ZM01"."209220CS22".TrfInSetBegin := NOT ("_PNComPLC308"."308210ZS01AccessStopRequest" AND NOT "_209220ZM01"."209220CS22".TrfInSetActive) AND "_209220ZM01Orders"."220CR21-220CS22-TrfInSet";
END_REGION

REGION Network 50: **** 5.2 - Equations - Flow Equation **** 220CS22 Transfer OUT Set Begin
   "_209220ZM01"."209220CS22".TrfOutSetBegin := NOT ("_DPComPLC212"."212AAccessStopRequest" AND NOT "_209220ZM01"."209220CS22".TrfOutSetActive) AND "_209220ZM01Orders"."220CS22-220CR23-TrfInSet";
END_REGION

REGION Network 51: **** 5.2 - Equations - Flow Equation **** 220CR23 Transfer IN Set Begin
   "_209220ZM01"."209220CR23".TrfInSetBegin := NOT ("_DPComPLC212"."212AAccessStopRequest" AND NOT "_209220ZM01"."209220CR23".TrfInSetActive) AND "_209220ZM01Orders"."220CS22-220CR23-TrfInSet";
END_REGION

REGION Network 52: **** 5.2 - Equations - Flow Equation **** 220CR23 Transfer OUT Set Begin
   "_209220ZM01"."209220CR23".TrfOutSetBegin := NOT ("_DPComPLC212"."212AAccessStopRequest" AND NOT "_209220ZM01"."209220CR23".TrfOutSetActive) AND "_209220ZM01Orders"."220CR23-R228.02-TrfOutSet";
END_REGION

REGION Network 53: **** 5.2 - Equations - Flow Equations *** Infeed wait condition
   // LineFeed - Infeed late condition
   "_209220ZM01"."209220CS22LineFeed".InfeedWaitCond := NOT "_PNComPLC308"."308220CR28".BodyInPosition AND NOT "_209220ZMS011Modes".EmptyStnModeSel AND NOT "_209220ZMS012Modes".EmptyStnModeSel;
END_REGION

REGION Network 54: **** 5.2 - Equations - Flow Equations ***Infeed wait late condition done
   // LineFeed - Infeed wait late condition done
   "_209220ZM01"."209220CS22LineFeed".InfeedWaitDoneCond := NOT "_209220ZM01"."209220CS22LineFeed".InfeedWaitCond OR "_209220ZMS011Modes".EmptyStnModeSel OR "_209220ZMS012Modes".EmptyStnModeSel;
END_REGION

REGION Network 55: **** 5.2 - Equations - Flow Equations ***Outfeed wait condition
   // LineFeed - Outfeed late condition
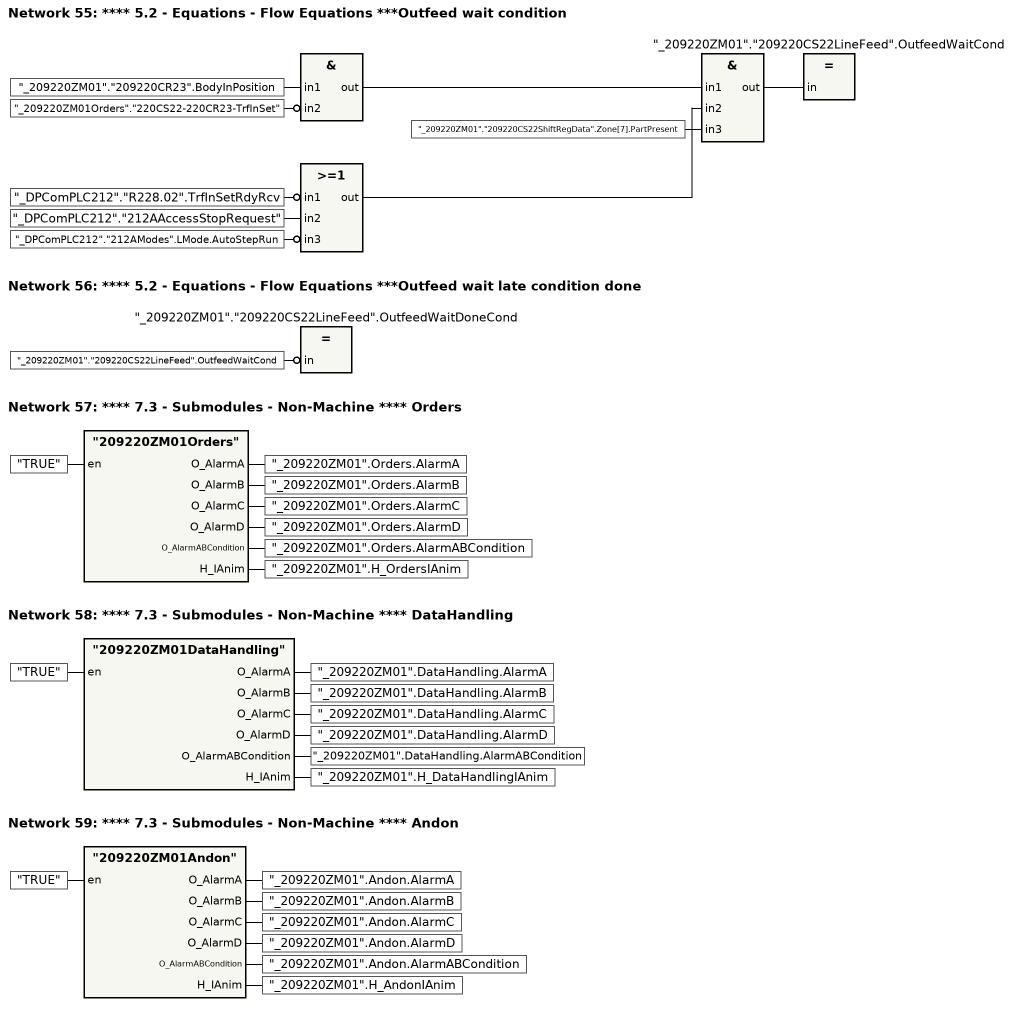
   "_209220ZM01"."209220CS22LineFeed".OutfeedWaitCond := "_209220ZM01"."209220CR23".BodyInPosition AND NOT "_209220ZM01Orders"."220CS22-220CR23-TrfInSet" AND (NOT "_DPComPLC212"."R228.02".TrfInSetRdyRcv OR "_DPComPLC212"."212AAccessStopRequest" OR NOT "_DPComPLC212"."212AModes".LMode.AutoStepRun) AND "_209220ZM01"."209220CS22ShiftRegData".Zone[7].PartPresent;
END_REGION

REGION Network 56: **** 5.2 - Equations - Flow Equations ***Outfeed wait late condition done
   // LineFeed - Outfeed wait late condition done
   "_209220ZM01"."209220CS22LineFeed".OutfeedWaitDoneCond := NOT "_209220ZM01"."209220CS22LineFeed".OutfeedWaitCond;
END_REGION

REGION Network 57: **** 7.3 - Submodules - Non-Machine **** Orders
   IF "TRUE" THEN
       "209220ZM01Orders"(O_AlarmA => "_209220ZM01".Orders.AlarmA,
                          O_AlarmB => "_209220ZM01".Orders.AlarmB,
                          O_AlarmC => "_209220ZM01".Orders.AlarmC,
                          O_AlarmD => "_209220ZM01".Orders.AlarmD,
                          O_AlarmABCondition => "_209220ZM01".Orders.AlarmABCondition,
                          H_IAnim => "_209220ZM01".H_OrdersIAnim);
   END_IF;
END_REGION

REGION Network 58: **** 7.3 - Submodules - Non-Machine **** DataHandling
   // Data Handling
   IF "TRUE" THEN
       "209220ZM01DataHandling"(O_AlarmA => "_209220ZM01".DataHandling.AlarmA,
                               O_AlarmB => "_209220ZM01".DataHandling.AlarmB,
                               O_AlarmC => "_209220ZM01".DataHandling.AlarmC,
                               O_AlarmD => "_209220ZM01".DataHandling.AlarmD,
                               O_AlarmABCondition => "_209220ZM01".DataHandling.AlarmABCondition,
                               H_IAnim => "_209220ZM01".H_DataHandlingIAnim);
   END_IF;
END_REGION

REGION Network 59: **** 7.3 - Submodules - Non-Machine **** Andon
   IF "TRUE" THEN
       "209220ZM01Andon"(O_AlarmA => "_209220ZM01".Andon.AlarmA,
                         O_AlarmB => "_209220ZM01".Andon.AlarmB,
                         O_AlarmC => "_209220ZM01".Andon.AlarmC,
                         O_AlarmD => "_209220ZM01".Andon.AlarmD,
                         O_AlarmABCondition => "_209220ZM01".Andon.AlarmABCondition,
                         H_IAnim => "_209220ZM01".H_AndonIAnim);
   END_IF;
END_REGION

REGION Network 60: **** 7.3 - Submodule - Machine **** 220CHB21
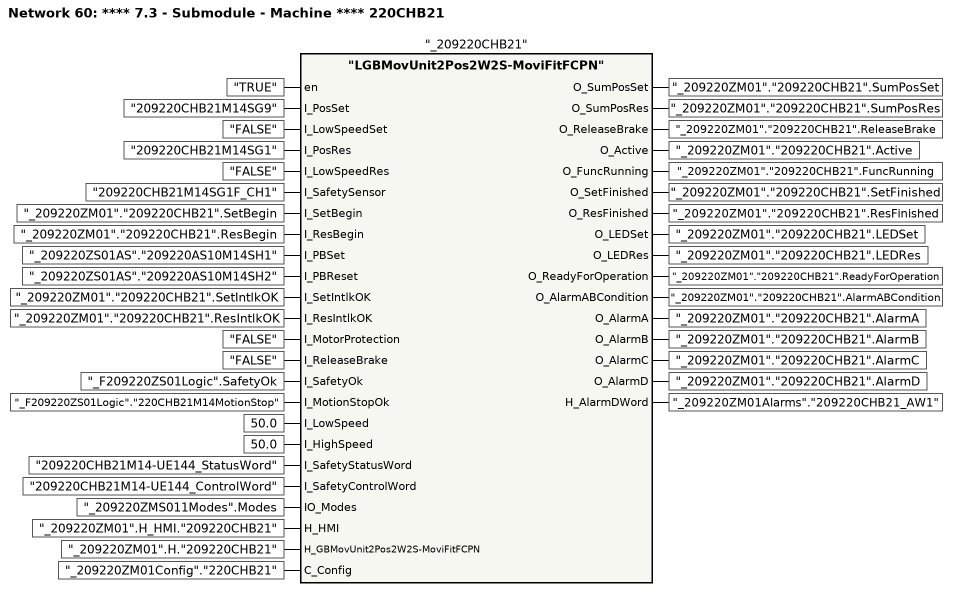
   IF "TRUE" THEN
       "_209220CHB21"(I_PosSet := "209220CHB21M14SG9",   // "LGBMovUnit2Pos2W2S-MoviFitFCPN"
                      I_LowSpeedSet := "FALSE",
                      I_PosRes := "209220CHB21M14SG1",
                      I_LowSpeedRes := "FALSE",
                      I_SafetySensor := "209220CHB21M14SG1F_CH1",
                      I_SetBegin := "_209220ZM01"."209220CHB21".SetBegin,
                      I_ResBegin := "_209220ZM01"."209220CHB21".ResBegin,
                      I_PBSet := "_209220ZS01AS"."209220AS10M14SH1",
                      I_PBReset := "_209220ZS01AS"."209220AS10M14SH2",
                      I_SetIntlkOK := "_209220ZM01"."209220CHB21".SetIntlkOK,
                      I_ResIntlkOK := "_209220ZM01"."209220CHB21".ResIntlkOK,
                      I_MotorProtection := "FALSE",
                      I_ReleaseBrake := "FALSE",
                      I_SafetyOk := "_F209220ZS01Logic".SafetyOk,
                      I_MotionStopOk := "_F209220ZS01Logic"."220CHB21M14MotionStop",
                      I_LowSpeed := 50.0,
                      I_HighSpeed := 50.0,
                      I_SafetyStatusWord := "209220CHB21M14-UE144_StatusWord",
                      I_SafetyControlWord := "209220CHB21M14-UE144_ControlWord",
                      IO_Modes := "_209220ZMS011Modes".Modes,
                      H_HMI := "_209220ZM01".H_HMI."209220CHB21",
                      "H_GBMovUnit2Pos2W2S-MoviFitFCPN" := "_209220ZM01".H."209220CHB21",
                      C_Config := "_209220ZM01Config"."220CHB21",
                      O_SumPosSet => "_209220ZM01"."209220CHB21".SumPosSet,
                      O_SumPosRes => "_209220ZM01"."209220CHB21".SumPosRes,
                      O_ReleaseBrake => "_209220ZM01"."209220CHB21".ReleaseBrake,
                      O_Active => "_209220ZM01"."209220CHB21".Active,
                      O_FuncRunning => "_209220ZM01"."209220CHB21".FuncRunning,
                      O_SetFinished => "_209220ZM01"."209220CHB21".SetFinished,
                      O_ResFinished => "_209220ZM01"."209220CHB21".ResFinished,
                      O_LEDSet => "_209220ZM01"."209220CHB21".LEDSet,
                      O_LEDRes => "_209220ZM01"."209220CHB21".LEDRes,
                      O_ReadyForOperation => "_209220ZM01"."209220CHB21".ReadyForOperation,
                      O_AlarmABCondition => "_209220ZM01"."209220CHB21".AlarmABCondition,
                      O_AlarmA => "_209220ZM01"."209220CHB21".AlarmA,
                      O_AlarmB => "_209220ZM01"."209220CHB21".AlarmB,
                      O_AlarmC => "_209220ZM01"."209220CHB21".AlarmC,
                      O_AlarmD => "_209220ZM01"."209220CHB21".AlarmD,
                      H_AlarmDWord => "_209220ZM01Alarms"."209220CHB21_AW1");
   END_IF;
END_REGION

REGION Network 61: **** 7.3 - Submodule - Machine **** 220CR21
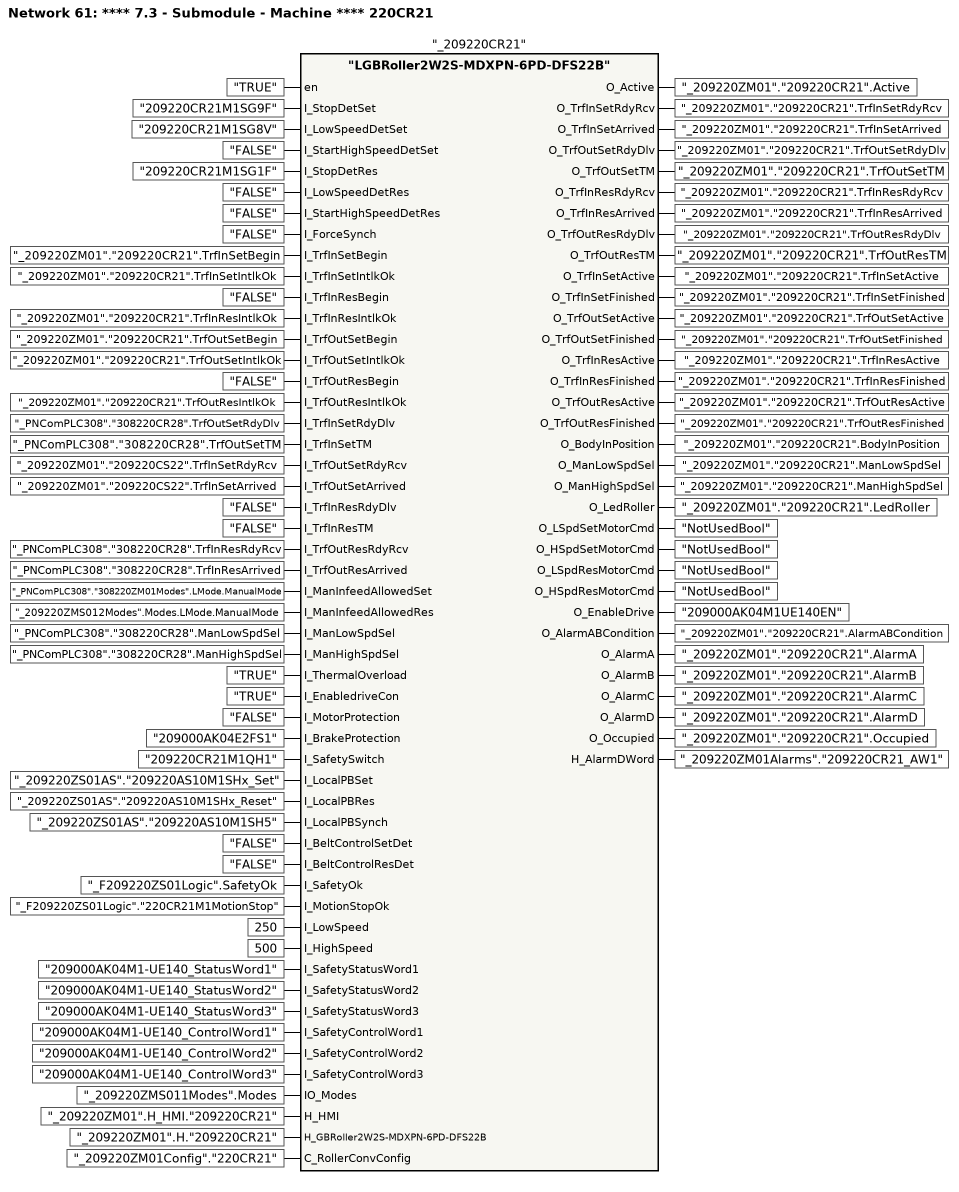
   IF "TRUE" THEN
       "_209220CR21"(I_StopDetSet := "209220CR21M1SG9F",   // "LGBRoller2W2S-MDXPN-6PD-DFS22B"
                     I_LowSpeedDetSet := "209220CR21M1SG8V",
                     I_StartHighSpeedDetSet := "FALSE",
                     I_StopDetRes := "209220CR21M1SG1F",
                     I_LowSpeedDetRes := "FALSE",
                     I_StartHighSpeedDetRes := "FALSE",
                     I_ForceSynch := "FALSE",
                     I_TrfInSetBegin := "_209220ZM01"."209220CR21".TrfInSetBegin,
                     I_TrfInSetIntlkOk := "_209220ZM01"."209220CR21".TrfInSetIntlkOk,
                     I_TrfInResBegin := "FALSE",
                     I_TrfInResIntlkOk := "_209220ZM01"."209220CR21".TrfInResIntlkOk,
                     I_TrfOutSetBegin := "_209220ZM01"."209220CR21".TrfOutSetBegin,
                     I_TrfOutSetIntlkOk := "_209220ZM01"."209220CR21".TrfOutSetIntlkOk,
                     I_TrfOutResBegin := "FALSE",
                     I_TrfOutResIntlkOk := "_209220ZM01"."209220CR21".TrfOutResIntlkOk,
                     I_TrfInSetRdyDlv := "_PNComPLC308"."308220CR28".TrfOutSetRdyDlv,
                     I_TrfInSetTM := "_PNComPLC308"."308220CR28".TrfOutSetTM,
                     I_TrfOutSetRdyRcv := "_209220ZM01"."209220CS22".TrfInSetRdyRcv,
                     I_TrfOutSetArrived := "_209220ZM01"."209220CS22".TrfInSetArrived,
                     I_TrfInResRdyDlv := "FALSE",
                     I_TrfInResTM := "FALSE",
                     I_TrfOutResRdyRcv := "_PNComPLC308"."308220CR28".TrfInResRdyRcv,
                     I_TrfOutResArrived := "_PNComPLC308"."308220CR28".TrfInResArrived,
                     I_ManInfeedAllowedSet := "_PNComPLC308"."308220ZM01Modes".LMode.ManualMode,
                     I_ManInfeedAllowedRes := "_209220ZMS012Modes".Modes.LMode.ManualMode,
                     I_ManLowSpdSel := "_PNComPLC308"."308220CR28".ManLowSpdSel,
                     I_ManHighSpdSel := "_PNComPLC308"."308220CR28".ManHighSpdSel,
                     I_ThermalOverload := "TRUE",
                     I_EnabledriveCon := "TRUE",
                     I_MotorProtection := "FALSE",
                     I_BrakeProtection := "209000AK04E2FS1",
                     I_SafetySwitch := "209220CR21M1QH1",
                     I_LocalPBSet := "_209220ZS01AS"."209220AS10M1SHx_Set",
                     I_LocalPBRes := "_209220ZS01AS"."209220AS10M1SHx_Reset",
                     I_LocalPBSynch := "_209220ZS01AS"."209220AS10M1SH5",
                     I_BeltControlSetDet := "FALSE",
                     I_BeltControlResDet := "FALSE",
                     I_SafetyOk := "_F209220ZS01Logic".SafetyOk,
                     I_MotionStopOk := "_F209220ZS01Logic"."220CR21M1MotionStop",
                     I_LowSpeed := 250,
                     I_HighSpeed := 500,
                     I_SafetyStatusWord1 := "209000AK04M1-UE140_StatusWord1",
                     I_SafetyStatusWord2 := "209000AK04M1-UE140_StatusWord2",
                     I_SafetyStatusWord3 := "209000AK04M1-UE140_StatusWord3",
                     I_SafetyControlWord1 := "209000AK04M1-UE140_ControlWord1",
                     I_SafetyControlWord2 := "209000AK04M1-UE140_ControlWord2",
                     I_SafetyControlWord3 := "209000AK04M1-UE140_ControlWord3",
                     IO_Modes := "_209220ZMS011Modes".Modes,
                     H_HMI := "_209220ZM01".H_HMI."209220CR21",
                     "H_GBRoller2W2S-MDXPN-6PD-DFS22B" := "_209220ZM01".H."209220CR21",
                     C_RollerConvConfig := "_209220ZM01Config"."220CR21",
                     O_Active => "_209220ZM01"."209220CR21".Active,
                     O_TrfInSetRdyRcv => "_209220ZM01"."209220CR21".TrfInSetRdyRcv,
                     O_TrfInSetArrived => "_209220ZM01"."209220CR21".TrfInSetArrived,
                     O_TrfOutSetRdyDlv => "_209220ZM01"."209220CR21".TrfOutSetRdyDlv,
                     O_TrfOutSetTM => "_209220ZM01"."209220CR21".TrfOutSetTM,
                     O_TrfInResRdyRcv => "_209220ZM01"."209220CR21".TrfInResRdyRcv,
                     O_TrfInResArrived => "_209220ZM01"."209220CR21".TrfInResArrived,
                     O_TrfOutResRdyDlv => "_209220ZM01"."209220CR21".TrfOutResRdyDlv,
                     O_TrfOutResTM => "_209220ZM01"."209220CR21".TrfOutResTM,
                     O_TrfInSetActive => "_209220ZM01"."209220CR21".TrfInSetActive,
                     O_TrfInSetFinished => "_209220ZM01"."209220CR21".TrfInSetFinished,
                     O_TrfOutSetActive => "_209220ZM01"."209220CR21".TrfOutSetActive,
                     O_TrfOutSetFinished => "_209220ZM01"."209220CR21".TrfOutSetFinished,
                     O_TrfInResActive => "_209220ZM01"."209220CR21".TrfInResActive,
                     O_TrfInResFinished => "_209220ZM01"."209220CR21".TrfInResFinished,
                     O_TrfOutResActive => "_209220ZM01"."209220CR21".TrfOutResActive,
                     O_TrfOutResFinished => "_209220ZM01"."209220CR21".TrfOutResFinished,
                     O_BodyInPosition => "_209220ZM01"."209220CR21".BodyInPosition,
                     O_ManLowSpdSel => "_209220ZM01"."209220CR21".ManLowSpdSel,
                     O_ManHighSpdSel => "_209220ZM01"."209220CR21".ManHighSpdSel,
                     O_LedRoller => "_209220ZM01"."209220CR21".LedRoller,
                     O_LSpdSetMotorCmd => "NotUsedBool",
                     O_HSpdSetMotorCmd => "NotUsedBool",
                     O_LSpdResMotorCmd => "NotUsedBool",
                     O_HSpdResMotorCmd => "NotUsedBool",
                     O_EnableDrive => "209000AK04M1UE140EN",
                     O_AlarmABCondition => "_209220ZM01"."209220CR21".AlarmABCondition,
                     O_AlarmA => "_209220ZM01"."209220CR21".AlarmA,
                     O_AlarmB => "_209220ZM01"."209220CR21".AlarmB,
                     O_AlarmC => "_209220ZM01"."209220CR21".AlarmC,
                     O_AlarmD => "_209220ZM01"."209220CR21".AlarmD,
                     O_Occupied => "_209220ZM01"."209220CR21".Occupied,
                     H_AlarmDWord => "_209220ZM01Alarms"."209220CR21_AW1");
   END_IF;
END_REGION

REGION Network 62: **** 7.3 - Submodule - Machine **** 220CS22
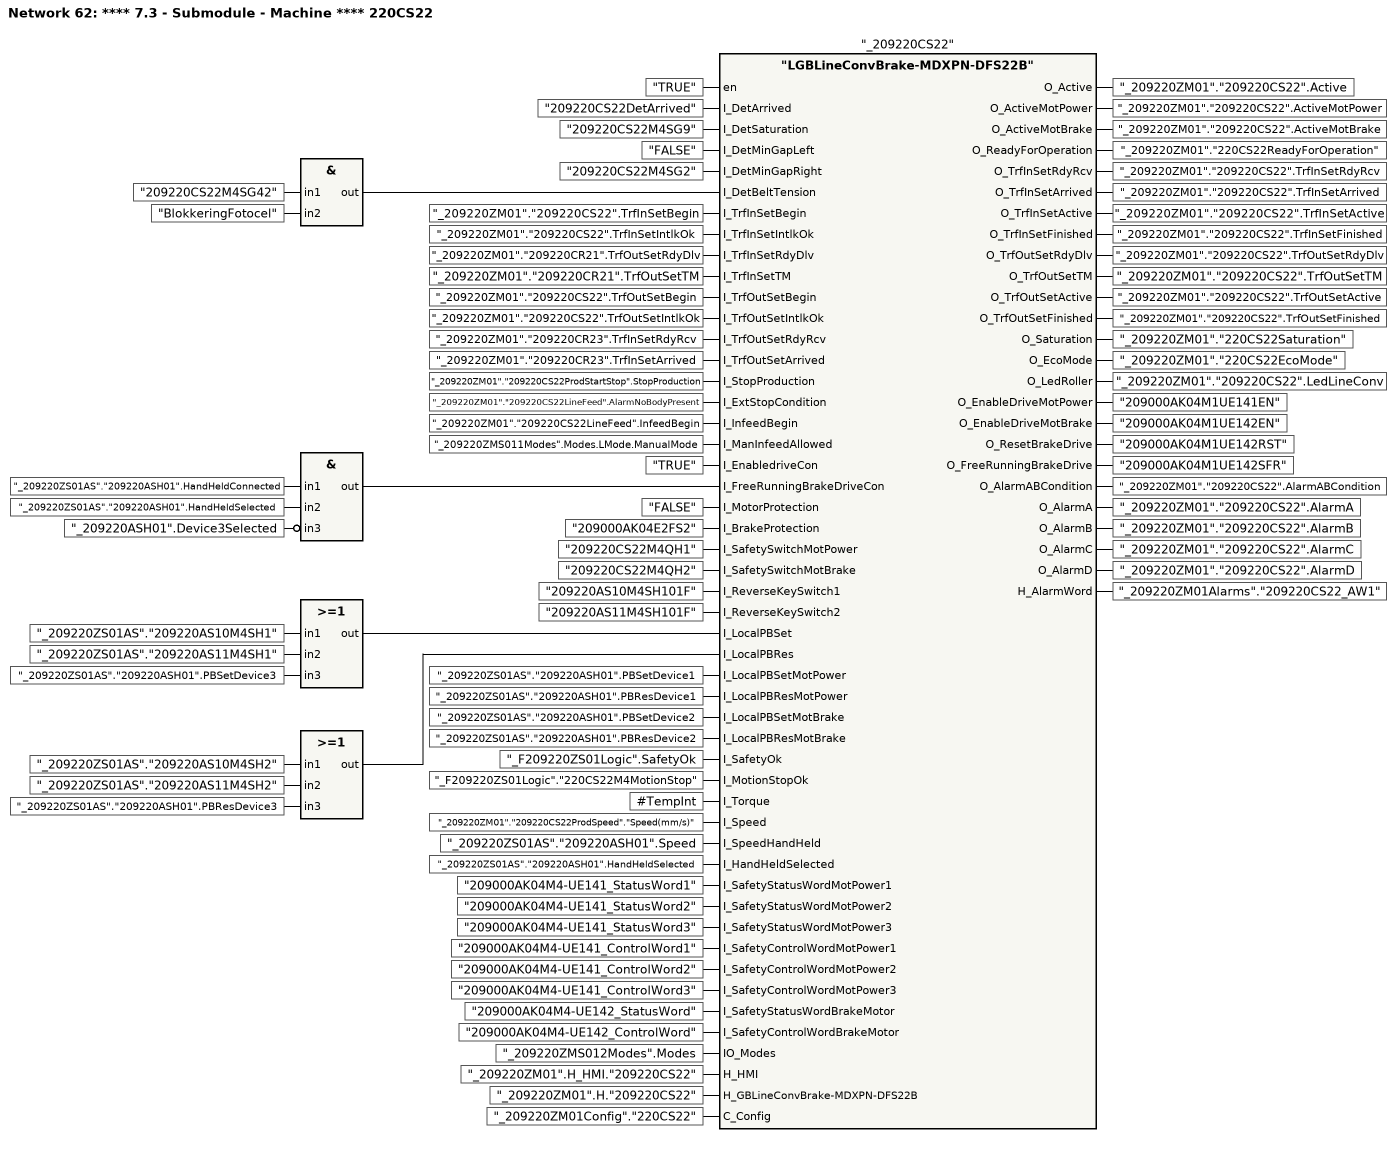
   IF "TRUE" THEN
       "_209220CS22"(I_DetArrived := "209220CS22DetArrived",   // "LGBLineConvBrake-MDXPN-DFS22B"
                     I_DetSaturation := "209220CS22M4SG9",
                     I_DetMinGapLeft := "FALSE",
                     I_DetMinGapRight := "209220CS22M4SG2",
                     I_DetBeltTension := "209220CS22M4SG42" AND "BlokkeringFotocel",
                     I_TrfInSetBegin := "_209220ZM01"."209220CS22".TrfInSetBegin,
                     I_TrfInSetIntlkOk := "_209220ZM01"."209220CS22".TrfInSetIntlkOk,
                     I_TrfInSetRdyDlv := "_209220ZM01"."209220CR21".TrfOutSetRdyDlv,
                     I_TrfInSetTM := "_209220ZM01"."209220CR21".TrfOutSetTM,
                     I_TrfOutSetBegin := "_209220ZM01"."209220CS22".TrfOutSetBegin,
                     I_TrfOutSetIntlkOk := "_209220ZM01"."209220CS22".TrfOutSetIntlkOk,
                     I_TrfOutSetRdyRcv := "_209220ZM01"."209220CR23".TrfInSetRdyRcv,
                     I_TrfOutSetArrived := "_209220ZM01"."209220CR23".TrfInSetArrived,
                     I_StopProduction := "_209220ZM01"."209220CS22ProdStartStop".StopProduction,
                     I_ExtStopCondition := "_209220ZM01"."209220CS22LineFeed".AlarmNoBodyPresent,
                     I_InfeedBegin := "_209220ZM01"."209220CS22LineFeed".InfeedBegin,
                     I_ManInfeedAllowed := "_209220ZMS011Modes".Modes.LMode.ManualMode,
                     I_EnabledriveCon := "TRUE",
                     I_FreeRunningBrakeDriveCon := "_209220ZS01AS"."209220ASH01".HandHeldConnected AND "_209220ZS01AS"."209220ASH01".HandHeldSelected AND NOT "_209220ASH01".Device3Selected,
                     I_MotorProtection := "FALSE",
                     I_BrakeProtection := "209000AK04E2FS2",
                     I_SafetySwitchMotPower := "209220CS22M4QH1",
                     I_SafetySwitchMotBrake := "209220CS22M4QH2",
                     I_ReverseKeySwitch1 := "209220AS10M4SH101F",
                     I_ReverseKeySwitch2 := "209220AS11M4SH101F",
                     I_LocalPBSet := "_209220ZS01AS"."209220AS10M4SH1" OR "_209220ZS01AS"."209220AS11M4SH1" OR "_209220ZS01AS"."209220ASH01".PBSetDevice3,
                     I_LocalPBRes := "_209220ZS01AS"."209220AS10M4SH2" OR "_209220ZS01AS"."209220AS11M4SH2" OR "_209220ZS01AS"."209220ASH01".PBResDevice3,
                     I_LocalPBSetMotPower := "_209220ZS01AS"."209220ASH01".PBSetDevice1,
                     I_LocalPBResMotPower := "_209220ZS01AS"."209220ASH01".PBResDevice1,
                     I_LocalPBSetMotBrake := "_209220ZS01AS"."209220ASH01".PBSetDevice2,
                     I_LocalPBResMotBrake := "_209220ZS01AS"."209220ASH01".PBResDevice2,
                     I_SafetyOk := "_F209220ZS01Logic".SafetyOk,
                     I_MotionStopOk := "_F209220ZS01Logic"."220CS22M4MotionStop",
                     I_Torque := #TempInt,
                     I_Speed := "_209220ZM01"."209220CS22ProdSpeed"."Speed(mm/s)",
                     I_SpeedHandHeld := "_209220ZS01AS"."209220ASH01".Speed,
                     I_HandHeldSelected := "_209220ZS01AS"."209220ASH01".HandHeldSelected,
                     I_SafetyStatusWordMotPower1 := "209000AK04M4-UE141_StatusWord1",
                     I_SafetyStatusWordMotPower2 := "209000AK04M4-UE141_StatusWord2",
                     I_SafetyStatusWordMotPower3 := "209000AK04M4-UE141_StatusWord3",
                     I_SafetyControlWordMotPower1 := "209000AK04M4-UE141_ControlWord1",
                     I_SafetyControlWordMotPower2 := "209000AK04M4-UE141_ControlWord2",
                     I_SafetyControlWordMotPower3 := "209000AK04M4-UE141_ControlWord3",
                     I_SafetyStatusWordBrakeMotor := "209000AK04M4-UE142_StatusWord",
                     I_SafetyControlWordBrakeMotor := "209000AK04M4-UE142_ControlWord",
                     IO_Modes := "_209220ZMS012Modes".Modes,
                     H_HMI := "_209220ZM01".H_HMI."209220CS22",
                     "H_GBLineConvBrake-MDXPN-DFS22B" := "_209220ZM01".H."209220CS22",
                     C_Config := "_209220ZM01Config"."220CS22",
                     O_Active => "_209220ZM01"."209220CS22".Active,
                     O_ActiveMotPower => "_209220ZM01"."209220CS22".ActiveMotPower,
                     O_ActiveMotBrake => "_209220ZM01"."209220CS22".ActiveMotBrake,
                     O_ReadyForOperation => "_209220ZM01"."220CS22ReadyForOperation",
                     O_TrfInSetRdyRcv => "_209220ZM01"."209220CS22".TrfInSetRdyRcv,
                     O_TrfInSetArrived => "_209220ZM01"."209220CS22".TrfInSetArrived,
                     O_TrfInSetActive => "_209220ZM01"."209220CS22".TrfInSetActive,
                     O_TrfInSetFinished => "_209220ZM01"."209220CS22".TrfInSetFinished,
                     O_TrfOutSetRdyDlv => "_209220ZM01"."209220CS22".TrfOutSetRdyDlv,
                     O_TrfOutSetTM => "_209220ZM01"."209220CS22".TrfOutSetTM,
                     O_TrfOutSetActive => "_209220ZM01"."209220CS22".TrfOutSetActive,
                     O_TrfOutSetFinished => "_209220ZM01"."209220CS22".TrfOutSetFinished,
                     O_Saturation => "_209220ZM01"."220CS22Saturation",
                     O_EcoMode => "_209220ZM01"."220CS22EcoMode",
                     O_LedRoller => "_209220ZM01"."209220CS22".LedLineConv,
                     O_EnableDriveMotPower => "209000AK04M1UE141EN",
                     O_EnableDriveMotBrake => "209000AK04M1UE142EN",
                     O_ResetBrakeDrive => "209000AK04M1UE142RST",
                     O_FreeRunningBrakeDrive => "209000AK04M1UE142SFR",
                     O_AlarmABCondition => "_209220ZM01"."209220CS22".AlarmABCondition,
                     O_AlarmA => "_209220ZM01"."209220CS22".AlarmA,
                     O_AlarmB => "_209220ZM01"."209220CS22".AlarmB,
                     O_AlarmC => "_209220ZM01"."209220CS22".AlarmC,
                     O_AlarmD => "_209220ZM01"."209220CS22".AlarmD,
                     H_AlarmWord => "_209220ZM01Alarms"."209220CS22_AW1");
   END_IF;
END_REGION

REGION Network 63: **** 7.3 - Submodule - Machine **** 220CR23
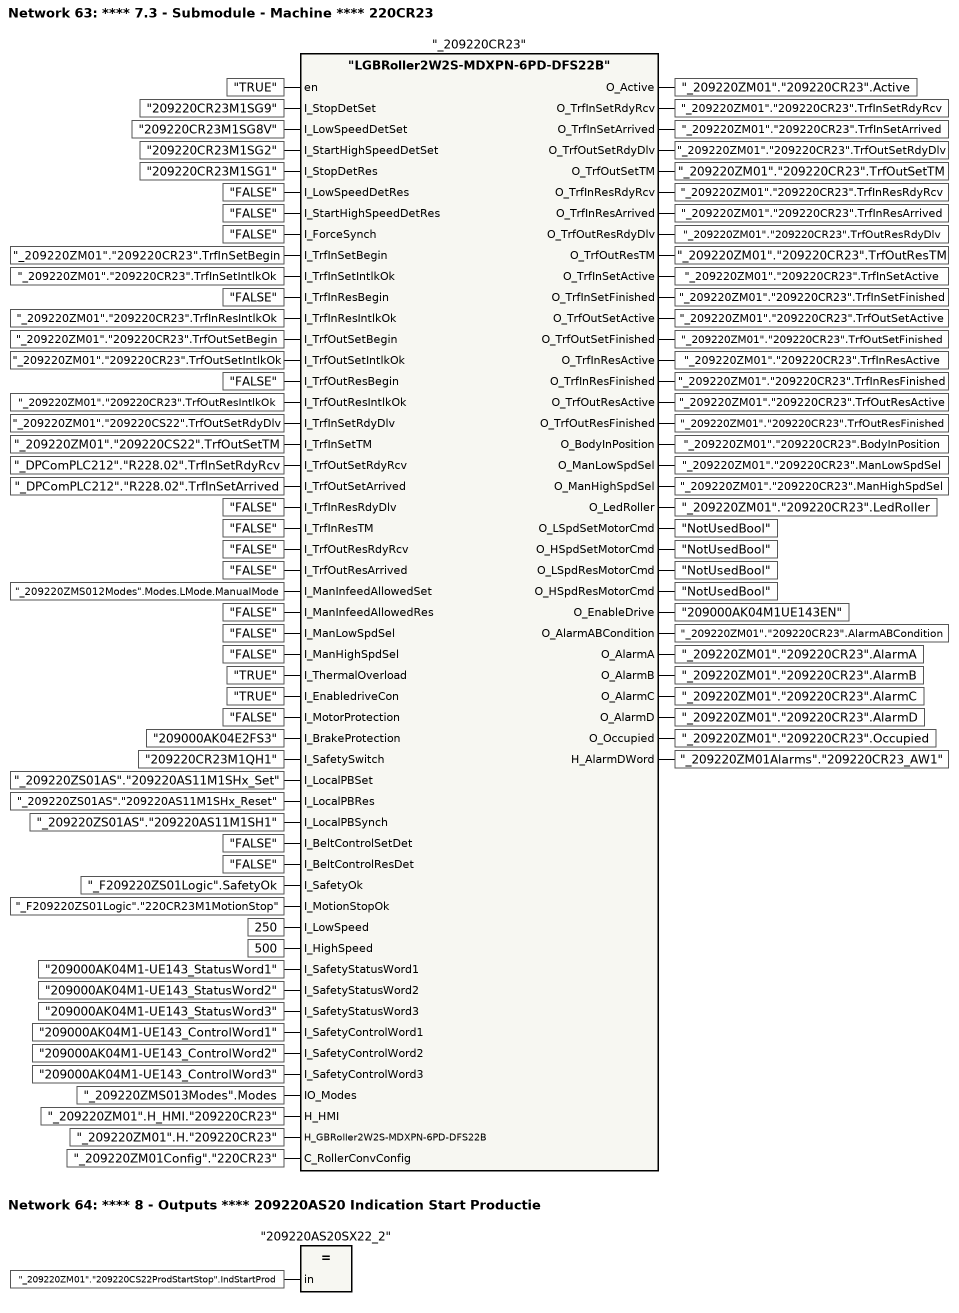
   IF "TRUE" THEN
       "_209220CR23"(I_StopDetSet := "209220CR23M1SG9",   // "LGBRoller2W2S-MDXPN-6PD-DFS22B"
                     I_LowSpeedDetSet := "209220CR23M1SG8V",
                     I_StartHighSpeedDetSet := "209220CR23M1SG2",
                     I_StopDetRes := "209220CR23M1SG1",
                     I_LowSpeedDetRes := "FALSE",
                     I_StartHighSpeedDetRes := "FALSE",
                     I_ForceSynch := "FALSE",
                     I_TrfInSetBegin := "_209220ZM01"."209220CR23".TrfInSetBegin,
                     I_TrfInSetIntlkOk := "_209220ZM01"."209220CR23".TrfInSetIntlkOk,
                     I_TrfInResBegin := "FALSE",
                     I_TrfInResIntlkOk := "_209220ZM01"."209220CR23".TrfInResIntlkOk,
                     I_TrfOutSetBegin := "_209220ZM01"."209220CR23".TrfOutSetBegin,
                     I_TrfOutSetIntlkOk := "_209220ZM01"."209220CR23".TrfOutSetIntlkOk,
                     I_TrfOutResBegin := "FALSE",
                     I_TrfOutResIntlkOk := "_209220ZM01"."209220CR23".TrfOutResIntlkOk,
                     I_TrfInSetRdyDlv := "_209220ZM01"."209220CS22".TrfOutSetRdyDlv,
                     I_TrfInSetTM := "_209220ZM01"."209220CS22".TrfOutSetTM,
                     I_TrfOutSetRdyRcv := "_DPComPLC212"."R228.02".TrfInSetRdyRcv,
                     I_TrfOutSetArrived := "_DPComPLC212"."R228.02".TrfInSetArrived,
                     I_TrfInResRdyDlv := "FALSE",
                     I_TrfInResTM := "FALSE",
                     I_TrfOutResRdyRcv := "FALSE",
                     I_TrfOutResArrived := "FALSE",
                     I_ManInfeedAllowedSet := "_209220ZMS012Modes".Modes.LMode.ManualMode,
                     I_ManInfeedAllowedRes := "FALSE",
                     I_ManLowSpdSel := "FALSE",
                     I_ManHighSpdSel := "FALSE",
                     I_ThermalOverload := "TRUE",
                     I_EnabledriveCon := "TRUE",
                     I_MotorProtection := "FALSE",
                     I_BrakeProtection := "209000AK04E2FS3",
                     I_SafetySwitch := "209220CR23M1QH1",
                     I_LocalPBSet := "_209220ZS01AS"."209220AS11M1SHx_Set",
                     I_LocalPBRes := "_209220ZS01AS"."209220AS11M1SHx_Reset",
                     I_LocalPBSynch := "_209220ZS01AS"."209220AS11M1SH1",
                     I_BeltControlSetDet := "FALSE",
                     I_BeltControlResDet := "FALSE",
                     I_SafetyOk := "_F209220ZS01Logic".SafetyOk,
                     I_MotionStopOk := "_F209220ZS01Logic"."220CR23M1MotionStop",
                     I_LowSpeed := 250,
                     I_HighSpeed := 500,
                     I_SafetyStatusWord1 := "209000AK04M1-UE143_StatusWord1",
                     I_SafetyStatusWord2 := "209000AK04M1-UE143_StatusWord2",
                     I_SafetyStatusWord3 := "209000AK04M1-UE143_StatusWord3",
                     I_SafetyControlWord1 := "209000AK04M1-UE143_ControlWord1",
                     I_SafetyControlWord2 := "209000AK04M1-UE143_ControlWord2",
                     I_SafetyControlWord3 := "209000AK04M1-UE143_ControlWord3",
                     IO_Modes := "_209220ZMS013Modes".Modes,
                     H_HMI := "_209220ZM01".H_HMI."209220CR23",
                     "H_GBRoller2W2S-MDXPN-6PD-DFS22B" := "_209220ZM01".H."209220CR23",
                     C_RollerConvConfig := "_209220ZM01Config"."220CR23",
                     O_Active => "_209220ZM01"."209220CR23".Active,
                     O_TrfInSetRdyRcv => "_209220ZM01"."209220CR23".TrfInSetRdyRcv,
                     O_TrfInSetArrived => "_209220ZM01"."209220CR23".TrfInSetArrived,
                     O_TrfOutSetRdyDlv => "_209220ZM01"."209220CR23".TrfOutSetRdyDlv,
                     O_TrfOutSetTM => "_209220ZM01"."209220CR23".TrfOutSetTM,
                     O_TrfInResRdyRcv => "_209220ZM01"."209220CR23".TrfInResRdyRcv,
                     O_TrfInResArrived => "_209220ZM01"."209220CR23".TrfInResArrived,
                     O_TrfOutResRdyDlv => "_209220ZM01"."209220CR23".TrfOutResRdyDlv,
                     O_TrfOutResTM => "_209220ZM01"."209220CR23".TrfOutResTM,
                     O_TrfInSetActive => "_209220ZM01"."209220CR23".TrfInSetActive,
                     O_TrfInSetFinished => "_209220ZM01"."209220CR23".TrfInSetFinished,
                     O_TrfOutSetActive => "_209220ZM01"."209220CR23".TrfOutSetActive,
                     O_TrfOutSetFinished => "_209220ZM01"."209220CR23".TrfOutSetFinished,
                     O_TrfInResActive => "_209220ZM01"."209220CR23".TrfInResActive,
                     O_TrfInResFinished => "_209220ZM01"."209220CR23".TrfInResFinished,
                     O_TrfOutResActive => "_209220ZM01"."209220CR23".TrfOutResActive,
                     O_TrfOutResFinished => "_209220ZM01"."209220CR23".TrfOutResFinished,
                     O_BodyInPosition => "_209220ZM01"."209220CR23".BodyInPosition,
                     O_ManLowSpdSel => "_209220ZM01"."209220CR23".ManLowSpdSel,
                     O_ManHighSpdSel => "_209220ZM01"."209220CR23".ManHighSpdSel,
                     O_LedRoller => "_209220ZM01"."209220CR23".LedRoller,
                     O_LSpdSetMotorCmd => "NotUsedBool",
                     O_HSpdSetMotorCmd => "NotUsedBool",
                     O_LSpdResMotorCmd => "NotUsedBool",
                     O_HSpdResMotorCmd => "NotUsedBool",
                     O_EnableDrive => "209000AK04M1UE143EN",
                     O_AlarmABCondition => "_209220ZM01"."209220CR23".AlarmABCondition,
                     O_AlarmA => "_209220ZM01"."209220CR23".AlarmA,
                     O_AlarmB => "_209220ZM01"."209220CR23".AlarmB,
                     O_AlarmC => "_209220ZM01"."209220CR23".AlarmC,
                     O_AlarmD => "_209220ZM01"."209220CR23".AlarmD,
                     O_Occupied => "_209220ZM01"."209220CR23".Occupied,
                     H_AlarmDWord => "_209220ZM01Alarms"."209220CR23_AW1");
   END_IF;
END_REGION

REGION Network 64: **** 8 - Outputs **** 209220AS20 Indication Start Productie
   "209220AS20SX22_2" := "_209220ZM01"."209220CS22ProdStartStop".IndStartProd;
END_REGION

REGION Network 65: **** 8 - Outputs **** 209220AS20 Indication Leegloop
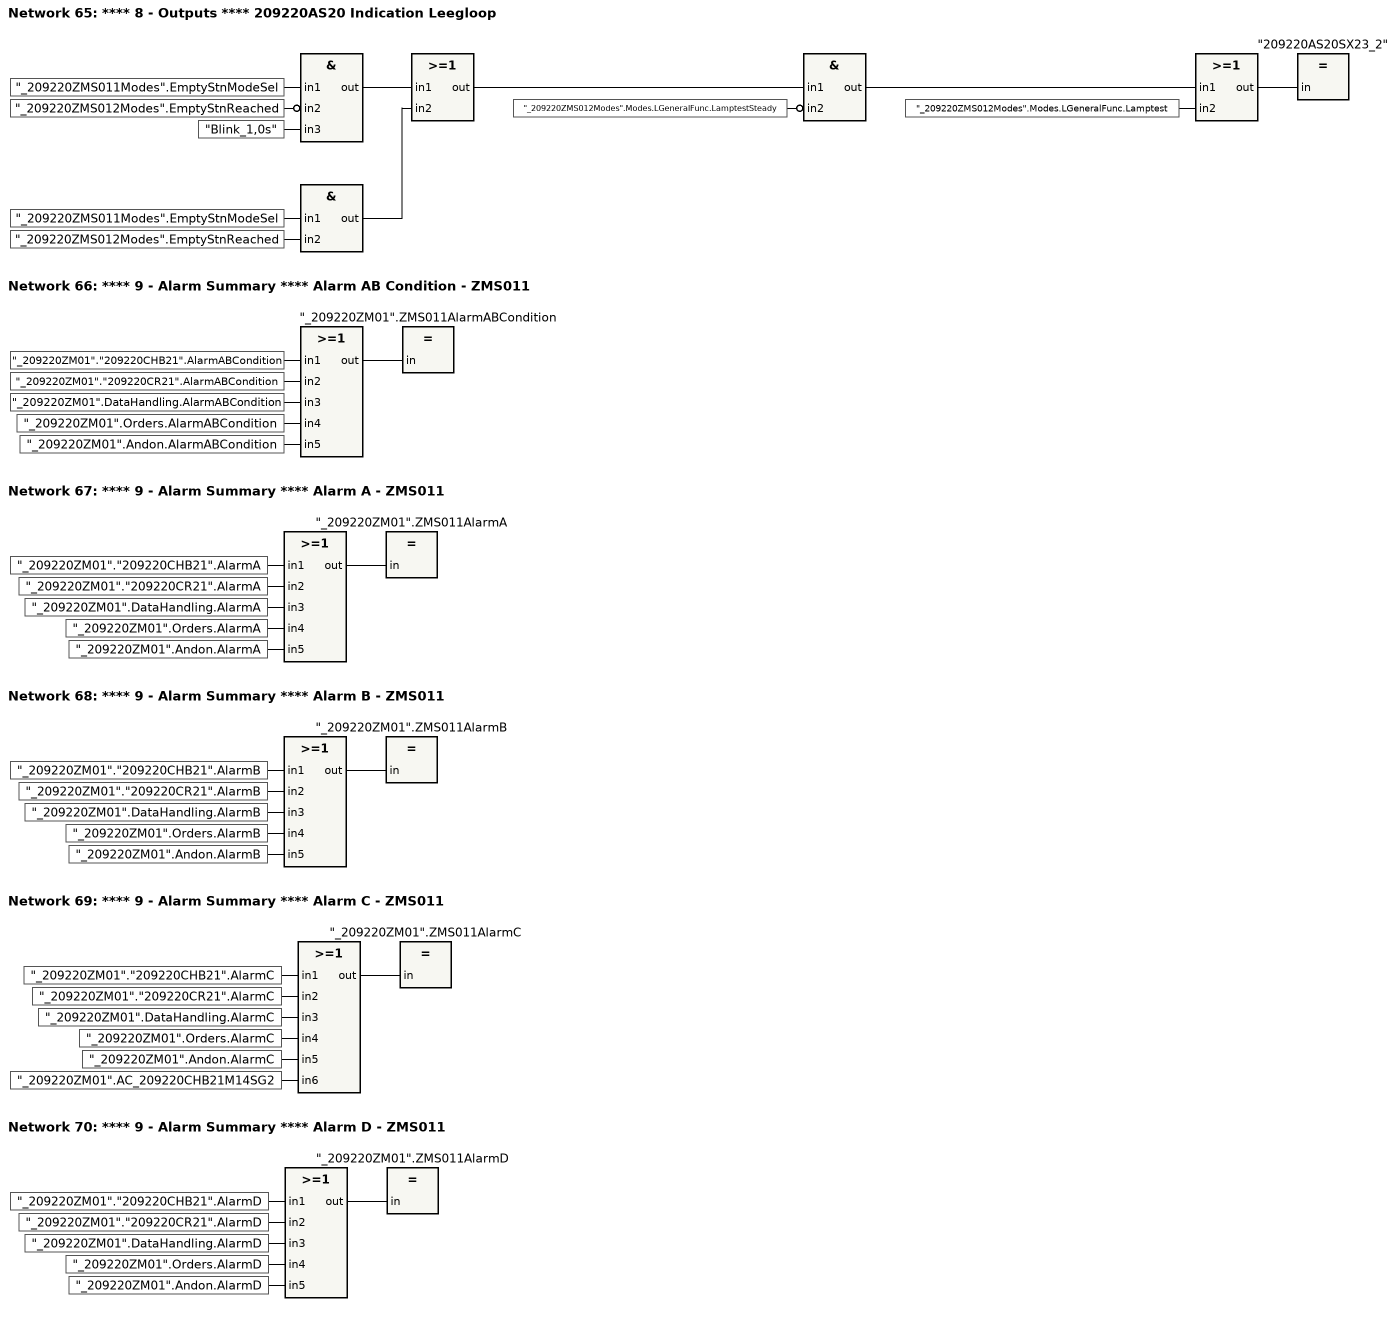
   "209220AS20SX23_2" := ((("_209220ZMS011Modes".EmptyStnModeSel AND NOT "_209220ZMS012Modes".EmptyStnReached AND "Blink_1,0s") OR ("_209220ZMS011Modes".EmptyStnModeSel AND "_209220ZMS012Modes".EmptyStnReached)) AND NOT "_209220ZMS012Modes".Modes.LGeneralFunc.LamptestSteady) OR "_209220ZMS012Modes".Modes.LGeneralFunc.Lamptest;
END_REGION

REGION Network 66: **** 9 - Alarm Summary **** Alarm AB Condition - ZMS011
   // Alarm AB condition
   "_209220ZM01".ZMS011AlarmABCondition := "_209220ZM01"."209220CHB21".AlarmABCondition OR "_209220ZM01"."209220CR21".AlarmABCondition OR "_209220ZM01".DataHandling.AlarmABCondition OR "_209220ZM01".Orders.AlarmABCondition OR "_209220ZM01".Andon.AlarmABCondition;
END_REGION

REGION Network 67: **** 9 - Alarm Summary **** Alarm A - ZMS011
   // Summary of alarms A
   "_209220ZM01".ZMS011AlarmA := "_209220ZM01"."209220CHB21".AlarmA OR "_209220ZM01"."209220CR21".AlarmA OR "_209220ZM01".DataHandling.AlarmA OR "_209220ZM01".Orders.AlarmA OR "_209220ZM01".Andon.AlarmA;
END_REGION

REGION Network 68: **** 9 - Alarm Summary **** Alarm B - ZMS011
   // Summary of alarms B
   "_209220ZM01".ZMS011AlarmB := "_209220ZM01"."209220CHB21".AlarmB OR "_209220ZM01"."209220CR21".AlarmB OR "_209220ZM01".DataHandling.AlarmB OR "_209220ZM01".Orders.AlarmB OR "_209220ZM01".Andon.AlarmB;
END_REGION

REGION Network 69: **** 9 - Alarm Summary **** Alarm C - ZMS011
   // Summary of alarms C
   "_209220ZM01".ZMS011AlarmC := "_209220ZM01"."209220CHB21".AlarmC OR "_209220ZM01"."209220CR21".AlarmC OR "_209220ZM01".DataHandling.AlarmC OR "_209220ZM01".Orders.AlarmC OR "_209220ZM01".Andon.AlarmC OR "_209220ZM01".AC_209220CHB21M14SG2;
END_REGION

REGION Network 70: **** 9 - Alarm Summary **** Alarm D - ZMS011
   // Summary of alarms D
   "_209220ZM01".ZMS011AlarmD := "_209220ZM01"."209220CHB21".AlarmD OR "_209220ZM01"."209220CR21".AlarmD OR "_209220ZM01".DataHandling.AlarmD OR "_209220ZM01".Orders.AlarmD OR "_209220ZM01".Andon.AlarmD;
END_REGION

REGION Network 71: **** 9 - Alarm Summary **** Alarm AB Condition - ZMS012
   // Alarm AB condition
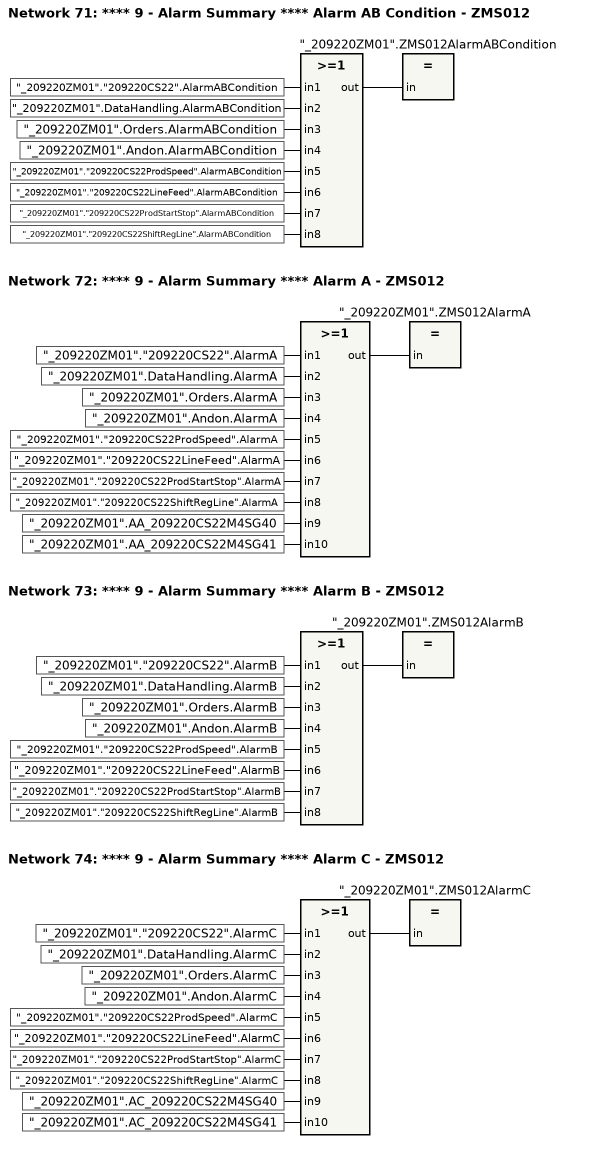
   "_209220ZM01".ZMS012AlarmABCondition := "_209220ZM01"."209220CS22".AlarmABCondition OR "_209220ZM01".DataHandling.AlarmABCondition OR "_209220ZM01".Orders.AlarmABCondition OR "_209220ZM01".Andon.AlarmABCondition OR "_209220ZM01"."209220CS22ProdSpeed".AlarmABCondition OR "_209220ZM01"."209220CS22LineFeed".AlarmABCondition OR "_209220ZM01"."209220CS22ProdStartStop".AlarmABCondition OR "_209220ZM01"."209220CS22ShiftRegLine".AlarmABCondition;
END_REGION

REGION Network 72: **** 9 - Alarm Summary **** Alarm A - ZMS012
   // Summary of alarms A
   "_209220ZM01".ZMS012AlarmA := "_209220ZM01"."209220CS22".AlarmA OR "_209220ZM01".DataHandling.AlarmA OR "_209220ZM01".Orders.AlarmA OR "_209220ZM01".Andon.AlarmA OR "_209220ZM01"."209220CS22ProdSpeed".AlarmA OR "_209220ZM01"."209220CS22LineFeed".AlarmA OR "_209220ZM01"."209220CS22ProdStartStop".AlarmA OR "_209220ZM01"."209220CS22ShiftRegLine".AlarmA OR "_209220ZM01".AA_209220CS22M4SG40 OR "_209220ZM01".AA_209220CS22M4SG41;
END_REGION

REGION Network 73: **** 9 - Alarm Summary **** Alarm B - ZMS012
   // Summary of alarms B
   "_209220ZM01".ZMS012AlarmB := "_209220ZM01"."209220CS22".AlarmB OR "_209220ZM01".DataHandling.AlarmB OR "_209220ZM01".Orders.AlarmB OR "_209220ZM01".Andon.AlarmB OR "_209220ZM01"."209220CS22ProdSpeed".AlarmB OR "_209220ZM01"."209220CS22LineFeed".AlarmB OR "_209220ZM01"."209220CS22ProdStartStop".AlarmB OR "_209220ZM01"."209220CS22ShiftRegLine".AlarmB;
END_REGION

REGION Network 74: **** 9 - Alarm Summary **** Alarm C - ZMS012
   // Summary of alarms C
   "_209220ZM01".ZMS012AlarmC := "_209220ZM01"."209220CS22".AlarmC OR "_209220ZM01".DataHandling.AlarmC OR "_209220ZM01".Orders.AlarmC OR "_209220ZM01".Andon.AlarmC OR "_209220ZM01"."209220CS22ProdSpeed".AlarmC OR "_209220ZM01"."209220CS22LineFeed".AlarmC OR "_209220ZM01"."209220CS22ProdStartStop".AlarmC OR "_209220ZM01"."209220CS22ShiftRegLine".AlarmC OR "_209220ZM01".AC_209220CS22M4SG40 OR "_209220ZM01".AC_209220CS22M4SG41;
END_REGION

REGION Network 75: **** 9 - Alarm Summary **** Alarm D - ZMS012
   // Summary of alarms D
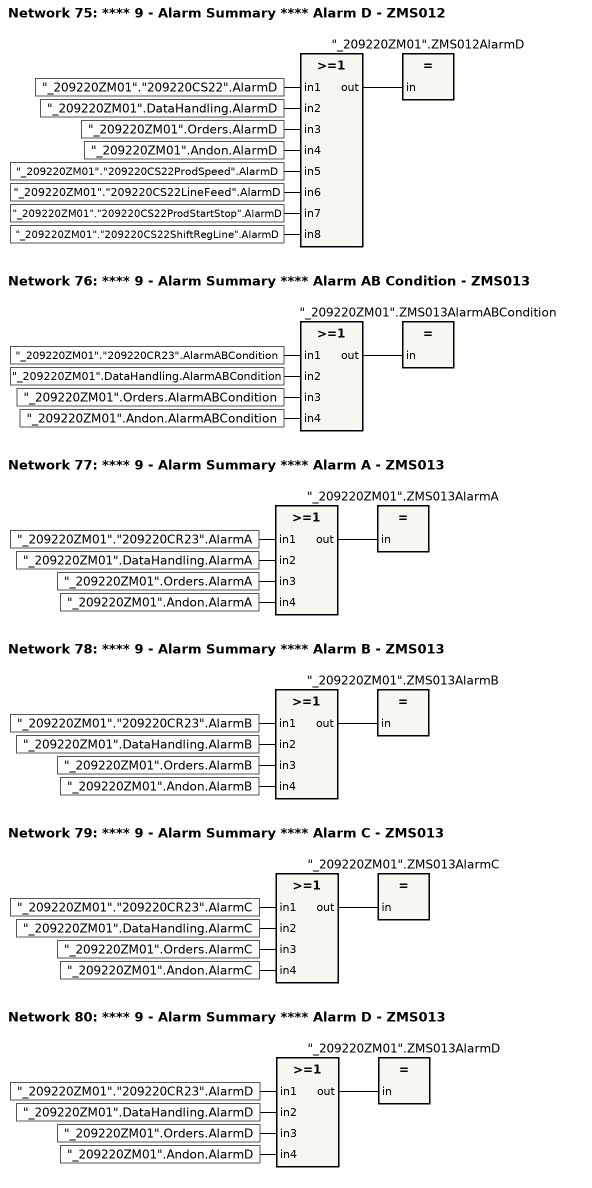
   "_209220ZM01".ZMS012AlarmD := "_209220ZM01"."209220CS22".AlarmD OR "_209220ZM01".DataHandling.AlarmD OR "_209220ZM01".Orders.AlarmD OR "_209220ZM01".Andon.AlarmD OR "_209220ZM01"."209220CS22ProdSpeed".AlarmD OR "_209220ZM01"."209220CS22LineFeed".AlarmD OR "_209220ZM01"."209220CS22ProdStartStop".AlarmD OR "_209220ZM01"."209220CS22ShiftRegLine".AlarmD;
END_REGION

REGION Network 76: **** 9 - Alarm Summary **** Alarm AB Condition - ZMS013
   // Alarm AB condition
   "_209220ZM01".ZMS013AlarmABCondition := "_209220ZM01"."209220CR23".AlarmABCondition OR "_209220ZM01".DataHandling.AlarmABCondition OR "_209220ZM01".Orders.AlarmABCondition OR "_209220ZM01".Andon.AlarmABCondition;
END_REGION

REGION Network 77: **** 9 - Alarm Summary **** Alarm A - ZMS013
   // Summary of alarms A
   "_209220ZM01".ZMS013AlarmA := "_209220ZM01"."209220CR23".AlarmA OR "_209220ZM01".DataHandling.AlarmA OR "_209220ZM01".Orders.AlarmA OR "_209220ZM01".Andon.AlarmA;
END_REGION

REGION Network 78: **** 9 - Alarm Summary **** Alarm B - ZMS013
   // Summary of alarms B
   "_209220ZM01".ZMS013AlarmB := "_209220ZM01"."209220CR23".AlarmB OR "_209220ZM01".DataHandling.AlarmB OR "_209220ZM01".Orders.AlarmB OR "_209220ZM01".Andon.AlarmB;
END_REGION

REGION Network 79: **** 9 - Alarm Summary **** Alarm C - ZMS013
   // Summary of alarms C
   "_209220ZM01".ZMS013AlarmC := "_209220ZM01"."209220CR23".AlarmC OR "_209220ZM01".DataHandling.AlarmC OR "_209220ZM01".Orders.AlarmC OR "_209220ZM01".Andon.AlarmC;
END_REGION

REGION Network 80: **** 9 - Alarm Summary **** Alarm D - ZMS013
   // Summary of alarms D
   "_209220ZM01".ZMS013AlarmD := "_209220ZM01"."209220CR23".AlarmD OR "_209220ZM01".DataHandling.AlarmD OR "_209220ZM01".Orders.AlarmD OR "_209220ZM01".Andon.AlarmD;
END_REGION

REGION Network 81: **** 9 - Alarm Summary **** Alarm AB Condition
   // Alarm AB condition
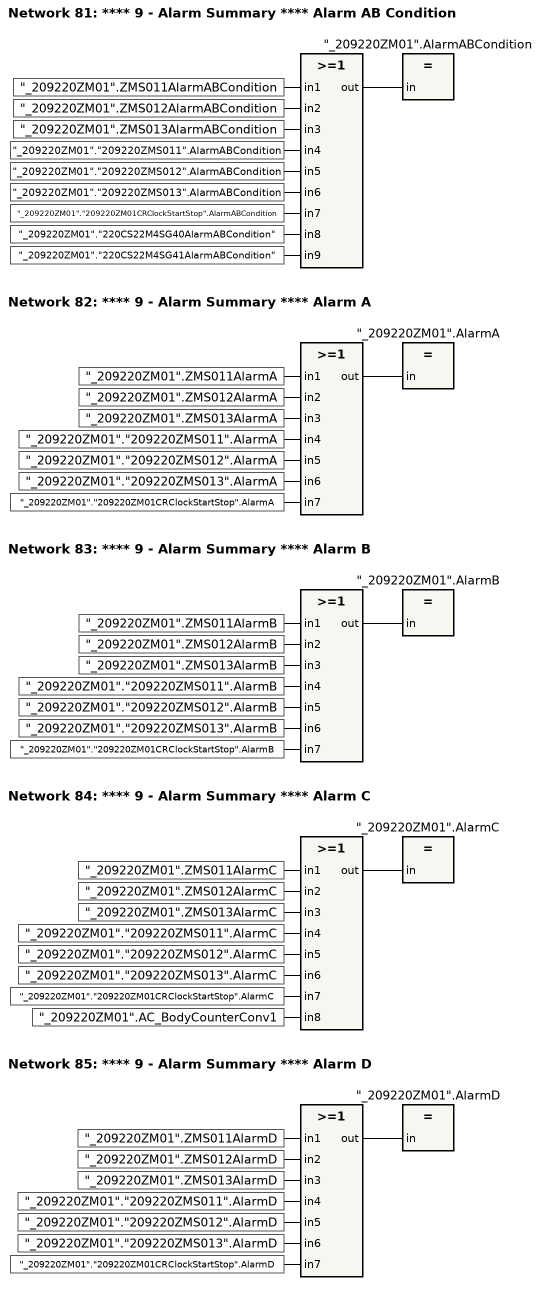
   "_209220ZM01".AlarmABCondition := "_209220ZM01".ZMS011AlarmABCondition OR "_209220ZM01".ZMS012AlarmABCondition OR "_209220ZM01".ZMS013AlarmABCondition OR "_209220ZM01"."209220ZMS011".AlarmABCondition OR "_209220ZM01"."209220ZMS012".AlarmABCondition OR "_209220ZM01"."209220ZMS013".AlarmABCondition OR "_209220ZM01"."209220ZM01CRClockStartStop".AlarmABCondition OR "_209220ZM01"."220CS22M4SG40AlarmABCondition" OR "_209220ZM01"."220CS22M4SG41AlarmABCondition";
END_REGION

REGION Network 82: **** 9 - Alarm Summary **** Alarm A
   // Summary of alarms A
   "_209220ZM01".AlarmA := "_209220ZM01".ZMS011AlarmA OR "_209220ZM01".ZMS012AlarmA OR "_209220ZM01".ZMS013AlarmA OR "_209220ZM01"."209220ZMS011".AlarmA OR "_209220ZM01"."209220ZMS012".AlarmA OR "_209220ZM01"."209220ZMS013".AlarmA OR "_209220ZM01"."209220ZM01CRClockStartStop".AlarmA;
END_REGION

REGION Network 83: **** 9 - Alarm Summary **** Alarm B
   // Summary of alarms B
   "_209220ZM01".AlarmB := "_209220ZM01".ZMS011AlarmB OR "_209220ZM01".ZMS012AlarmB OR "_209220ZM01".ZMS013AlarmB OR "_209220ZM01"."209220ZMS011".AlarmB OR "_209220ZM01"."209220ZMS012".AlarmB OR "_209220ZM01"."209220ZMS013".AlarmB OR "_209220ZM01"."209220ZM01CRClockStartStop".AlarmB;
END_REGION

REGION Network 84: **** 9 - Alarm Summary **** Alarm C
   // Summary of alarms C
   "_209220ZM01".AlarmC := "_209220ZM01".ZMS011AlarmC OR "_209220ZM01".ZMS012AlarmC OR "_209220ZM01".ZMS013AlarmC OR "_209220ZM01"."209220ZMS011".AlarmC OR "_209220ZM01"."209220ZMS012".AlarmC OR "_209220ZM01"."209220ZMS013".AlarmC OR "_209220ZM01"."209220ZM01CRClockStartStop".AlarmC OR "_209220ZM01".AC_BodyCounterConv1;
END_REGION

REGION Network 85: **** 9 - Alarm Summary **** Alarm D
   // Summary of alarms D
   "_209220ZM01".AlarmD := "_209220ZM01".ZMS011AlarmD OR "_209220ZM01".ZMS012AlarmD OR "_209220ZM01".ZMS013AlarmD OR "_209220ZM01"."209220ZMS011".AlarmD OR "_209220ZM01"."209220ZMS012".AlarmD OR "_209220ZM01"."209220ZMS013".AlarmD OR "_209220ZM01"."209220ZM01CRClockStartStop".AlarmD;
END_REGION

REGION Network 86: **** 9.1 - Alarm Output **** Alarm AB condition
   // Alarm AB condition
